LIN {X 0,Y 343.887,Z 716.045,A -85,B 0,C 180,E1 -14281.046,E2 -14281.046} C_VEL
LIN {X 0,Y 344.919,Z 706.382,A -85,B 0,C 180,E1 -14282.219,E2 -14282.219} C_VEL
LIN {X 0,Y 345.964,Z 694.644,A -85,B 0,C 180,E1 -14283.359,E2 -14283.359} C_VEL
LIN {X 0,Y 346.283,Z 691.22,A -85,B 0,C 180,E1 -14283.642,E2 -14283.642} C_VEL
LIN {X 0,Y 344.349,Z 679.11,A -85,B 0,C 180,E1 -14284.621,E2 -14284.621} C_VEL
LIN {X 0,Y 341.376,Z 665.612,A -85,B 0,C 180,E1 -14285.494,E2 -14285.494} C_VEL
LIN {X 0,Y 339.656,Z 658.402,A -85,B 0,C 180,E1 -14285.879,E2 -14285.879} C_VEL
LIN {X 0,Y 339.842,Z 654.272,A -85,B 0,C 180,E1 -14289.417,E2 -14289.417} C_VEL
LIN {X 0,Y 340.111,Z 649.95,A -85,B 0,C 180,E1 -14293.184,E2 -14293.184} C_VEL
LIN {X 0,Y 340.493,Z 645.812,A -85,B 0,C 180,E1 -14296.876,E2 -14296.876} C_VEL
LIN {X 0,Y 340.727,Z 642.044,A -85,B 0,C 180,E1 -14300.502,E2 -14300.502} C_VEL
LIN {X 0,Y 341.051,Z 642.005,A -85,B 0,C 180,E1 -14302.897,E2 -14302.897} C_VEL
LIN {X 0,Y 341.173,Z 641.984,A -85,B 0,C 180,E1 -14307.638,E2 -14307.638} C_VEL
LIN {X 0,Y 341.3,Z 641.968,A -85,B 0,C 180,E1 -14310,E2 -14310} C_VEL
LIN {X 0,Y 341.172,Z 641.985,A -85,B 0,C 180,E1 -14312.361,E2 -14312.361} C_VEL
LIN {X 0,Y 341.028,Z 642.002,A -85,B 0,C 180,E1 -14315.914,E2 -14315.914} C_VEL
LIN {X 0,Y 340.866,Z 642.023,A -85,B 0,C 180,E1 -14318.298,E2 -14318.298} C_VEL
LIN {X 0,Y 340.336,Z 642.088,A -85,B 0,C 180,E1 -14321.917,E2 -14321.917} C_VEL
LIN {X 0,Y 340.189,Z 642.443,A -85,B 0,C 180,E1 -14322.528,E2 -14322.528} C_VEL
LIN {X 0,Y 339.825,Z 648.464,A -85,B 0,C 180,E1 -14326.83,E2 -14326.83} C_VEL
LIN {X 0,Y 339.592,Z 653.752,A -85,B 0,C 180,E1 -14330.598,E2 -14330.598} C_VEL
LIN {X 0,Y 339.509,Z 657.449,A -85,B 0,C 180,E1 -14333.241,E2 -14333.241} C_VEL
LIN {X 0,Y 342.868,Z 671.995,A -85,B 0,C 180,E1 -14334.04,E2 -14334.04} C_VEL
LIN {X 0,Y 345.151,Z 683.532,A -85,B 0,C 180,E1 -14334.867,E2 -14334.867} C_VEL
LIN {X 0,Y 346.164,Z 690.83,A -85,B 0,C 180,E1 -14335.477,E2 -14335.477} C_VEL
LIN {X 0,Y 345.207,Z 701.967,A -85,B 0,C 180,E1 -14336.467,E2 -14336.467} C_VEL
LIN {X 0,Y 344.102,Z 712.788,A -85,B 0,C 180,E1 -14337.687,E2 -14337.687} C_VEL
LIN {X 0,Y 342.966,Z 723.402,A -85,B 0,C 180,E1 -14339.183,E2 -14339.183} C_VEL
LIN {X 0,Y 341.993,Z 731.641,A -85,B 0,C 180,E1 -14340.609,E2 -14340.609} C_VEL
LIN {X 0,Y 341.029,Z 740,A -85,B 0,C 180,E1 -14342.398,E2 -14342.398} C_VEL
LIN {X 0,Y 340.265,Z 747.036,A -85,B 0,C 180,E1 -14344.291,E2 -14344.291} C_VEL
LIN {X 0,Y 339.695,Z 752.623,A -85,B 0,C 180,E1 -14346.208,E2 -14346.208} C_VEL
LIN {X 0,Y 339.249,Z 757.368,A -85,B 0,C 180,E1 -14348.424,E2 -14348.424} C_VEL
LIN {X 0,Y 338.966,Z 759.987,A -85,B 0,C 180,E1 -14350.18,E2 -14350.18} C_VEL
LIN {X 0,Y 338.177,Z 761.122,A -85,B 0,C 180,E1 -14351.156,E2 -14351.156} C_VEL
LIN {X 0,Y 335.209,Z 762.337,A -85,B 0,C 180,E1 -14352.752,E2 -14352.752} C_VEL
LIN {X 0,Y 332.789,Z 762.794,A -85,B 0,C 180,E1 -14354.052,E2 -14354.052} C_VEL
LIN {X 0,Y 331.794,Z 762.817,A -85,B 0,C 180,E1 -14355.061,E2 -14355.061} C_VEL
LIN {X 0,Y 331.734,Z 762.729,A -85,B 0,C 180,E1 -14355.402,E2 -14355.402} C_VEL
LIN {X 0,Y 331.941,Z 761.386,A -85,B 0,C 180,E1 -14357.819,E2 -14357.819} C_VEL
LIN {X 0,Y 332.191,Z 759.33,A -85,B 0,C 180,E1 -14359.607,E2 -14359.607} C_VEL
LIN {X 0,Y 332.629,Z 756.285,A -85,B 0,C 180,E1 -14361.421,E2 -14361.421} C_VEL
LIN {X 0,Y 333.184,Z 752.093,A -85,B 0,C 180,E1 -14363.277,E2 -14363.277} C_VEL
LIN {X 0,Y 334.084,Z 745.842,A -85,B 0,C 180,E1 -14365.39,E2 -14365.39} C_VEL
LIN {X 0,Y 335.2,Z 738.06,A -85,B 0,C 180,E1 -14367.407,E2 -14367.407} C_VEL
LIN {X 0,Y 336.361,Z 730.689,A -85,B 0,C 180,E1 -14368.942,E2 -14368.942} C_VEL
LIN {X 0,Y 337.701,Z 721.438,A -85,B 0,C 180,E1 -14370.522,E2 -14370.522} C_VEL
LIN {X 0,Y 339.034,Z 711.873,A -85,B 0,C 180,E1 -14371.838,E2 -14371.838} C_VEL
LIN {X 0,Y 340.374,Z 700.364,A -85,B 0,C 180,E1 -14373.111,E2 -14373.111} C_VEL
LIN {X 0,Y 341.026,Z 692.815,A -85,B 0,C 180,E1 -14373.804,E2 -14373.804} C_VEL
LIN {X 0,Y 339.014,Z 680.497,A -85,B 0,C 180,E1 -14374.932,E2 -14374.932} C_VEL
LIN {X 0,Y 335.765,Z 667.742,A -85,B 0,C 180,E1 -14375.943,E2 -14375.943} C_VEL
LIN {X 0,Y 332.789,Z 658.389,A -85,B 0,C 180,E1 -14376.591,E2 -14376.591} C_VEL
LIN {X 0,Y 332.987,Z 653.339,A -85,B 0,C 180,E1 -14380.263,E2 -14380.263} C_VEL
LIN {X 0,Y 333.147,Z 649.771,A -85,B 0,C 180,E1 -14382.822,E2 -14382.822} C_VEL
LIN {X 0,Y 333.525,Z 644.51,A -85,B 0,C 180,E1 -14386.597,E2 -14386.597} C_VEL
LIN {X 0,Y 333.508,Z 642.948,A -85,B 0,C 180,E1 -14387.835,E2 -14387.835} C_VEL
LIN {X 0,Y 333.925,Z 642.894,A -85,B 0,C 180,E1 -14391.563,E2 -14391.563} C_VEL
LIN {X 0,Y 334.012,Z 642.883,A -85,B 0,C 180,E1 -14393.961,E2 -14393.961} C_VEL
LIN {X 0,Y 334.104,Z 642.869,A -85,B 0,C 180,E1 -14397.589,E2 -14397.589} C_VEL
LIN {X 0,Y 334.264,Z 642.85,A -85,B 0,C 180,E1 -14400,E2 -14400} C_VEL
LIN {X 0,Y 334.104,Z 642.87,A -85,B 0,C 180,E1 -14402.411,E2 -14402.411} C_VEL
LIN {X 0,Y 334.022,Z 642.879,A -85,B 0,C 180,E1 -14407.253,E2 -14407.253} C_VEL
LIN {X 0,Y 333.83,Z 642.903,A -85,B 0,C 180,E1 -14410.922,E2 -14410.922} C_VEL
LIN {X 0,Y 333.804,Z 642.904,A -85,B 0,C 180,E1 -14414.634,E2 -14414.634} C_VEL
LIN {X 0,Y 333.793,Z 642.906,A -85,B 0,C 180,E1 -14418.656,E2 -14418.656} C_VEL
LIN {X 0,Y 333.689,Z 642.921,A -85,B 0,C 180,E1 -14422.278,E2 -14422.278} C_VEL
LIN {X 0,Y 333.733,Z 642.913,A -85,B 0,C 180,E1 -14426.247,E2 -14426.247} C_VEL
LIN {X 0,Y 333.708,Z 642.916,A -85,B 0,C 180,E1 -14428.972,E2 -14428.972} C_VEL
LIN {X 0,Y 333.64,Z 642.926,A -85,B 0,C 180,E1 -14432.587,E2 -14432.587} C_VEL
LIN {X 0,Y 333.674,Z 642.922,A -85,B 0,C 180,E1 -14436.139,E2 -14436.139} C_VEL
LIN {X 0,Y 333.644,Z 642.927,A -85,B 0,C 180,E1 -14439.193,E2 -14439.193} C_VEL
LIN {X 0,Y 333.63,Z 642.927,A -85,B 0,C 180,E1 -14442.501,E2 -14442.501} C_VEL
LIN {X 0,Y 333.699,Z 643.1,A -85,B 0,C 180,E1 -14446.659,E2 -14446.659} C_VEL
LIN {X 0,Y 334.54,Z 647.77,A -85,B 0,C 180,E1 -14450.154,E2 -14450.154} C_VEL
LIN {X 0,Y 335.04,Z 651.547,A -85,B 0,C 180,E1 -14452.855,E2 -14452.855} C_VEL
LIN {X 0,Y 335.093,Z 654.529,A -85,B 0,C 180,E1 -14454.881,E2 -14454.881} C_VEL
LIN {X 0,Y 334.469,Z 659.801,A -85,B 0,C 180,E1 -14458.312,E2 -14458.312} C_VEL
LIN {X 0,Y 334.02,Z 664.14,A -85,B 0,C 180,E1 -14461.058,E2 -14461.058} C_VEL
LIN {X 0,Y 333.409,Z 670.604,A -85,B 0,C 180,E1 -14465.066,E2 -14465.066} C_VEL
LIN {X 0,Y 333.052,Z 675.105,A -85,B 0,C 180,E1 -14467.763,E2 -14467.763} C_VEL
LIN {X 0,Y 336.355,Z 689.153,A -85,B 0,C 180,E1 -14468.626,E2 -14468.626} C_VEL
LIN {X 0,Y 338.206,Z 701.155,A -85,B 0,C 180,E1 -14469.526,E2 -14469.526} C_VEL
LIN {X 0,Y 339.301,Z 713.613,A -85,B 0,C 180,E1 -14470.646,E2 -14470.646} C_VEL
LIN {X 0,Y 339.303,Z 718.335,A -85,B 0,C 180,E1 -14471.117,E2 -14471.117} C_VEL
LIN {X 0,Y 337.949,Z 729.167,A -85,B 0,C 180,E1 -14472.294,E2 -14472.294} C_VEL
LIN {X 0,Y 336.552,Z 740.044,A -85,B 0,C 180,E1 -14473.798,E2 -14473.798} C_VEL
LIN {X 0,Y 335.251,Z 749.542,A -85,B 0,C 180,E1 -14475.431,E2 -14475.431} C_VEL
LIN {X 0,Y 334.107,Z 757.933,A -85,B 0,C 180,E1 -14477.241,E2 -14477.241} C_VEL
LIN {X 0,Y 333.243,Z 764.702,A -85,B 0,C 180,E1 -14479.059,E2 -14479.059} C_VEL
LIN {X 0,Y 332.621,Z 770.129,A -85,B 0,C 180,E1 -14480.883,E2 -14480.883} C_VEL
LIN {X 0,Y 332.157,Z 775.843,A -85,B 0,C 180,E1 -14483.318,E2 -14483.318} C_VEL
LIN {X 0,Y 332.012,Z 779.038,A -85,B 0,C 180,E1 -14485.143,E2 -14485.143} C_VEL
LIN {X 0,Y 332,Z 780.628,A -85,B 0,C 180,E1 -14486.359,E2 -14486.359} C_VEL
LIN {X 0,Y 331.916,Z 781.79,A -85,B 0,C 180,E1 -14487.573,E2 -14487.573} C_VEL
LIN {X 0,Y 331.925,Z 782.506,A -85,B 0,C 180,E1 -14488.787,E2 -14488.787} C_VEL
LIN {X 0,Y 331.972,Z 782.827,A -85,B 0,C 180,E1 -14490.001,E2 -14490.001} C_VEL
LIN {X 0,Y 331.922,Z 782.752,A -85,B 0,C 180,E1 -14491.214,E2 -14491.214} C_VEL
LIN {X 0,Y 331.914,Z 782.275,A -85,B 0,C 180,E1 -14492.428,E2 -14492.428} C_VEL
LIN {X 0,Y 331.998,Z 781.36,A -85,B 0,C 180,E1 -14493.642,E2 -14493.642} C_VEL
LIN {X 0,Y 332.1,Z 778.315,A -85,B 0,C 180,E1 -14496.074,E2 -14496.074} C_VEL
LIN {X 0,Y 332.377,Z 774.864,A -85,B 0,C 180,E1 -14497.9,E2 -14497.9} C_VEL
LIN {X 0,Y 332.83,Z 770.338,A -85,B 0,C 180,E1 -14499.726,E2 -14499.726} C_VEL
LIN {X 0,Y 333.53,Z 764.63,A -85,B 0,C 180,E1 -14501.548,E2 -14501.548} C_VEL
LIN {X 0,Y 334.595,Z 757.51,A -85,B 0,C 180,E1 -14503.359,E2 -14503.359} C_VEL
LIN {X 0,Y 335.905,Z 748.669,A -85,B 0,C 180,E1 -14505.161,E2 -14505.161} C_VEL
LIN {X 0,Y 337.134,Z 738.987,A -85,B 0,C 180,E1 -14506.766,E2 -14506.766} C_VEL
LIN {X 0,Y 338.547,Z 728.563,A -85,B 0,C 180,E1 -14508.143,E2 -14508.143} C_VEL
LIN {X 0,Y 339.976,Z 717.451,A -85,B 0,C 180,E1 -14509.315,E2 -14509.315} C_VEL
LIN {X 0,Y 339.221,Z 705.114,A -85,B 0,C 180,E1 -14510.483,E2 -14510.483} C_VEL
LIN {X 0,Y 337.175,Z 692.156,A -85,B 0,C 180,E1 -14511.525,E2 -14511.525} C_VEL
LIN {X 0,Y 334.348,Z 680.067,A -85,B 0,C 180,E1 -14512.349,E2 -14512.349} C_VEL
LIN {X 0,Y 333.232,Z 675.513,A -85,B 0,C 180,E1 -14512.642,E2 -14512.642} C_VEL
LIN {X 0,Y 333.811,Z 668.75,A -85,B 0,C 180,E1 -14516.915,E2 -14516.915} C_VEL
LIN {X 0,Y 334.465,Z 663.296,A -85,B 0,C 180,E1 -14520.512,E2 -14520.512} C_VEL
LIN {X 0,Y 334.971,Z 659.603,A -85,B 0,C 180,E1 -14523.059,E2 -14523.059} C_VEL
LIN {X 0,Y 335.311,Z 655.648,A -85,B 0,C 180,E1 -14525.936,E2 -14525.936} C_VEL
LIN {X 0,Y 335.104,Z 651.672,A -85,B 0,C 180,E1 -14529.105,E2 -14529.105} C_VEL
LIN {X 0,Y 334.499,Z 647.664,A -85,B 0,C 180,E1 -14532.662,E2 -14532.662} C_VEL
LIN {X 0,Y 333.883,Z 644.312,A -85,B 0,C 180,E1 -14536.002,E2 -14536.002} C_VEL
LIN {X 0,Y 333.643,Z 642.928,A -85,B 0,C 180,E1 -14537.619,E2 -14537.619} C_VEL
LIN {X 0,Y 333.654,Z 642.927,A -85,B 0,C 180,E1 -14541.202,E2 -14541.202} C_VEL
LIN {X 0,Y 333.678,Z 642.924,A -85,B 0,C 180,E1 -14543.861,E2 -14543.861} C_VEL
LIN {X 0,Y 333.645,Z 642.925,A -85,B 0,C 180,E1 -14547.413,E2 -14547.413} C_VEL
LIN {X 0,Y 333.692,Z 642.92,A -85,B 0,C 180,E1 -14551.026,E2 -14551.026} C_VEL
LIN {X 0,Y 333.737,Z 642.911,A -85,B 0,C 180,E1 -14553.754,E2 -14553.754} C_VEL
LIN {X 0,Y 333.721,Z 642.917,A -85,B 0,C 180,E1 -14557.914,E2 -14557.914} C_VEL
LIN {X 0,Y 333.796,Z 642.908,A -85,B 0,C 180,E1 -14561.59,E2 -14561.59} C_VEL
LIN {X 0,Y 333.81,Z 642.907,A -85,B 0,C 180,E1 -14565.577,E2 -14565.577} C_VEL
LIN {X 0,Y 333.836,Z 642.903,A -85,B 0,C 180,E1 -14569.078,E2 -14569.078} C_VEL
LIN {X 0,Y 334.027,Z 642.878,A -85,B 0,C 180,E1 -14572.748,E2 -14572.748} C_VEL
LIN {X 0,Y 333.813,Z 642.906,A -85,B 0,C 180,E1 -14575.169,E2 -14575.169} C_VEL
LIN {X 0,Y 334.107,Z 642.867,A -85,B 0,C 180,E1 -14577.589,E2 -14577.589} C_VEL
LIN {X 0,Y 334.249,Z 642.851,A -85,B 0,C 180,E1 -14580,E2 -14580} C_VEL
LIN {X 0,Y 334.109,Z 642.871,A -85,B 0,C 180,E1 -14582.411,E2 -14582.411} C_VEL
LIN {X 0,Y 333.851,Z 642.903,A -85,B 0,C 180,E1 -14583.621,E2 -14583.621} C_VEL
LIN {X 0,Y 333.874,Z 643.33,A -85,B 0,C 180,E1 -14584.83,E2 -14584.83} C_VEL
LIN {X 0,Y 334.288,Z 645.219,A -85,B 0,C 180,E1 -14587.247,E2 -14587.247} C_VEL
LIN {X 0,Y 334.222,Z 647.299,A -85,B 0,C 180,E1 -14589.685,E2 -14589.685} C_VEL
LIN {X 0,Y 333.822,Z 650.713,A -85,B 0,C 180,E1 -14593.39,E2 -14593.39} C_VEL
LIN {X 0,Y 333.411,Z 654.396,A -85,B 0,C 180,E1 -14597.164,E2 -14597.164} C_VEL
LIN {X 0,Y 333.052,Z 658.348,A -85,B 0,C 180,E1 -14601.022,E2 -14601.022} C_VEL
LIN {X 0,Y 332.945,Z 659.916,A -85,B 0,C 180,E1 -14602.454,E2 -14602.454} C_VEL
LIN {X 0,Y 334.924,Z 665.893,A -85,B 0,C 180,E1 -14602.866,E2 -14602.866} C_VEL
LIN {X 0,Y 338.155,Z 677.169,A -85,B 0,C 180,E1 -14603.746,E2 -14603.746} C_VEL
LIN {X 0,Y 340.197,Z 686.586,A -85,B 0,C 180,E1 -14604.577,E2 -14604.577} C_VEL
LIN {X 0,Y 341.253,Z 694.62,A -85,B 0,C 180,E1 -14605.356,E2 -14605.356} C_VEL
LIN {X 0,Y 339.972,Z 705.362,A -85,B 0,C 180,E1 -14606.389,E2 -14606.389} C_VEL
LIN {X 0,Y 338.659,Z 715.933,A -85,B 0,C 180,E1 -14607.667,E2 -14607.667} C_VEL
LIN {X 0,Y 337.213,Z 725.82,A -85,B 0,C 180,E1 -14609.159,E2 -14609.159} C_VEL
LIN {X 0,Y 335.819,Z 735.103,A -85,B 0,C 180,E1 -14610.902,E2 -14610.902} C_VEL
LIN {X 0,Y 334.778,Z 742.114,A -85,B 0,C 180,E1 -14612.532,E2 -14612.532} C_VEL
LIN {X 0,Y 333.856,Z 748.201,A -85,B 0,C 180,E1 -14614.272,E2 -14614.272} C_VEL
LIN {X 0,Y 333.081,Z 753.553,A -85,B 0,C 180,E1 -14616.214,E2 -14616.214} C_VEL
LIN {X 0,Y 332.489,Z 758.289,A -85,B 0,C 180,E1 -14618.547,E2 -14618.547} C_VEL
LIN {X 0,Y 332.005,Z 761.528,A -85,B 0,C 180,E1 -14621.012,E2 -14621.012} C_VEL
LIN {X 0,Y 331.866,Z 762.755,A -85,B 0,C 180,E1 -14622.662,E2 -14622.662} C_VEL
LIN {X 0,Y 331.753,Z 763.207,A -85,B 0,C 180,E1 -14624.354,E2 -14624.354} C_VEL
LIN {X 0,Y 331.756,Z 762.88,A -85,B 0,C 180,E1 -14626.077,E2 -14626.077} C_VEL
LIN {X 0,Y 331.862,Z 761.721,A -85,B 0,C 180,E1 -14627.835,E2 -14627.835} C_VEL
LIN {X 0,Y 332.08,Z 759.647,A -85,B 0,C 180,E1 -14629.631,E2 -14629.631} C_VEL
LIN {X 0,Y 332.375,Z 756.523,A -85,B 0,C 180,E1 -14631.477,E2 -14631.477} C_VEL
LIN {X 0,Y 332.922,Z 751.114,A -85,B 0,C 180,E1 -14633.766,E2 -14633.766} C_VEL
LIN {X 0,Y 333.541,Z 745.111,A -85,B 0,C 180,E1 -14635.691,E2 -14635.691} C_VEL
LIN {X 0,Y 334.396,Z 737.874,A -85,B 0,C 180,E1 -14637.519,E2 -14637.519} C_VEL
LIN {X 0,Y 335.431,Z 729.564,A -85,B 0,C 180,E1 -14639.209,E2 -14639.209} C_VEL
LIN {X 0,Y 336.509,Z 720.29,A -85,B 0,C 180,E1 -14640.747,E2 -14640.747} C_VEL
LIN {X 0,Y 337.656,Z 710.407,A -85,B 0,C 180,E1 -14642.075,E2 -14642.075} C_VEL
LIN {X 0,Y 338.721,Z 699.199,A -85,B 0,C 180,E1 -14643.282,E2 -14643.282} C_VEL
LIN {X 0,Y 339.263,Z 690.604,A -85,B 0,C 180,E1 -14644.048,E2 -14644.048} C_VEL
LIN {X 0,Y 337.079,Z 678.122,A -85,B 0,C 180,E1 -14645.071,E2 -14645.071} C_VEL
LIN {X 0,Y 334.142,Z 665.017,A -85,B 0,C 180,E1 -14645.93,E2 -14645.93} C_VEL
LIN {X 0,Y 332.598,Z 658.588,A -85,B 0,C 180,E1 -14646.292,E2 -14646.292} C_VEL
LIN {X 0,Y 332.831,Z 654.037,A -85,B 0,C 180,E1 -14650.253,E2 -14650.253} C_VEL
LIN {X 0,Y 333.131,Z 649.745,A -85,B 0,C 180,E1 -14654.082,E2 -14654.082} C_VEL
LIN {X 0,Y 333.411,Z 646.98,A -85,B 0,C 180,E1 -14656.592,E2 -14656.592} C_VEL
LIN {X 0,Y 333.666,Z 643.014,A -85,B 0,C 180,E1 -14660.299,E2 -14660.299} C_VEL
LIN {X 0,Y 333.994,Z 642.882,A -85,B 0,C 180,E1 -14662.746,E2 -14662.746} C_VEL
LIN {X 0,Y 333.812,Z 642.904,A -85,B 0,C 180,E1 -14665.169,E2 -14665.169} C_VEL
LIN {X 0,Y 334.11,Z 642.864,A -85,B 0,C 180,E1 -14667.588,E2 -14667.588} C_VEL
LIN {X 0,Y 334.251,Z 642.846,A -85,B 0,C 180,E1 -14669.999,E2 -14669.999} C_VEL
LIN {X 0,Y 334.11,Z 642.865,A -85,B 0,C 180,E1 -14672.411,E2 -14672.411} C_VEL
LIN {X 0,Y 333.999,Z 642.878,A -85,B 0,C 180,E1 -14676.039,E2 -14676.039} C_VEL
LIN {X 0,Y 333.787,Z 642.906,A -85,B 0,C 180,E1 -14678.475,E2 -14678.475} C_VEL
LIN {X 0,Y 333.187,Z 642.988,A -85,B 0,C 180,E1 -14682.292,E2 -14682.292} C_VEL
LIN {X 0,Y 332.798,Z 648.01,A -85,B 0,C 180,E1 -14685.934,E2 -14685.934} C_VEL
LIN {X 0,Y 332.662,Z 651.536,A -85,B 0,C 180,E1 -14688.475,E2 -14688.475} C_VEL
LIN {X 0,Y 332.434,Z 656.948,A -85,B 0,C 180,E1 -14692.366,E2 -14692.366} C_VEL
LIN {X 0,Y 332.45,Z 657.693,A -85,B 0,C 180,E1 -14692.857,E2 -14692.857} C_VEL
LIN {X 0,Y 335.759,Z 671.72,A -85,B 0,C 180,E1 -14693.638,E2 -14693.638} C_VEL
LIN {X 0,Y 338.216,Z 684.197,A -85,B 0,C 180,E1 -14694.556,E2 -14694.556} C_VEL
LIN {X 0,Y 339.313,Z 691.71,A -85,B 0,C 180,E1 -14695.207,E2 -14695.207} C_VEL
LIN {X 0,Y 338.268,Z 703.087,A -85,B 0,C 180,E1 -14696.257,E2 -14696.257} C_VEL
LIN {X 0,Y 337.023,Z 714.803,A -85,B 0,C 180,E1 -14697.644,E2 -14697.644} C_VEL
LIN {X 0,Y 335.884,Z 724.714,A -85,B 0,C 180,E1 -14699.109,E2 -14699.109} C_VEL
LIN {X 0,Y 334.75,Z 734.035,A -85,B 0,C 180,E1 -14700.83,E2 -14700.83} C_VEL
LIN {X 0,Y 333.858,Z 741.937,A -85,B 0,C 180,E1 -14702.644,E2 -14702.644} C_VEL
LIN {X 0,Y 333.077,Z 748.729,A -85,B 0,C 180,E1 -14704.623,E2 -14704.623} C_VEL
LIN {X 0,Y 332.501,Z 753.912,A -85,B 0,C 180,E1 -14706.563,E2 -14706.563} C_VEL
LIN {X 0,Y 332.149,Z 757.763,A -85,B 0,C 180,E1 -14708.474,E2 -14708.474} C_VEL
LIN {X 0,Y 331.848,Z 760.418,A -85,B 0,C 180,E1 -14710.322,E2 -14710.322} C_VEL
LIN {X 0,Y 331.678,Z 762.405,A -85,B 0,C 180,E1 -14712.691,E2 -14712.691} C_VEL
LIN {X 0,Y 331.719,Z 762.87,A -85,B 0,C 180,E1 -14714.358,E2 -14714.358} C_VEL
LIN {X 0,Y 331.734,Z 762.729,A -85,B 0,C 180,E1 -14715.402,E2 -14715.402} C_VEL
LIN {X 0,Y 331.141,Z 762.46,A -85,B 0,C 180,E1 -14716.416,E2 -14716.416} C_VEL
LIN {X 0,Y 328.43,Z 761.437,A -85,B 0,C 180,E1 -14718.064,E2 -14718.064} C_VEL
LIN {X 0,Y 326.193,Z 760.057,A -85,B 0,C 180,E1 -14719.384,E2 -14719.384} C_VEL
LIN {X 0,Y 325.35,Z 758.678,A -85,B 0,C 180,E1 -14720.389,E2 -14720.389} C_VEL
LIN {X 0,Y 325.346,Z 758.123,A -85,B 0,C 180,E1 -14720.725,E2 -14720.725} C_VEL
LIN {X 0,Y 325.989,Z 753.834,A -85,B 0,C 180,E1 -14722.908,E2 -14722.908} C_VEL
LIN {X 0,Y 326.729,Z 748.798,A -85,B 0,C 180,E1 -14724.823,E2 -14724.823} C_VEL
LIN {X 0,Y 327.748,Z 742.304,A -85,B 0,C 180,E1 -14726.749,E2 -14726.749} C_VEL
LIN {X 0,Y 329.093,Z 734.103,A -85,B 0,C 180,E1 -14728.673,E2 -14728.673} C_VEL
LIN {X 0,Y 330.429,Z 725.241,A -85,B 0,C 180,E1 -14730.347,E2 -14730.347} C_VEL
LIN {X 0,Y 331.967,Z 714.941,A -85,B 0,C 180,E1 -14731.897,E2 -14731.897} C_VEL
LIN {X 0,Y 333.399,Z 704.029,A -85,B 0,C 180,E1 -14733.219,E2 -14733.219} C_VEL
LIN {X 0,Y 334.446,Z 694.487,A -85,B 0,C 180,E1 -14734.149,E2 -14734.149} C_VEL
LIN {X 0,Y 332.802,Z 683.728,A -85,B 0,C 180,E1 -14735.2,E2 -14735.2} C_VEL
LIN {X 0,Y 329.742,Z 670.964,A -85,B 0,C 180,E1 -14736.278,E2 -14736.278} C_VEL
LIN {X 0,Y 325.783,Z 658.559,A -85,B 0,C 180,E1 -14737.222,E2 -14737.222} C_VEL
LIN {X 0,Y 326.081,Z 652.738,A -85,B 0,C 180,E1 -14741.498,E2 -14741.498} C_VEL
LIN {X 0,Y 326.42,Z 647.051,A -85,B 0,C 180,E1 -14745.664,E2 -14745.664} C_VEL
LIN {X 0,Y 326.503,Z 643.819,A -85,B 0,C 180,E1 -14748.122,E2 -14748.122} C_VEL
LIN {X 0,Y 326.867,Z 643.773,A -85,B 0,C 180,E1 -14751.508,E2 -14751.508} C_VEL
LIN {X 0,Y 326.986,Z 643.758,A -85,B 0,C 180,E1 -14753.831,E2 -14753.831} C_VEL
LIN {X 0,Y 327.045,Z 643.748,A -85,B 0,C 180,E1 -14757.537,E2 -14757.537} C_VEL
LIN {X 0,Y 327.215,Z 643.728,A -85,B 0,C 180,E1 -14760,E2 -14760} C_VEL
LIN {X 0,Y 327.045,Z 643.749,A -85,B 0,C 180,E1 -14762.463,E2 -14762.463} C_VEL
LIN {X 0,Y 326.993,Z 643.754,A -85,B 0,C 180,E1 -14766.169,E2 -14766.169} C_VEL
LIN {X 0,Y 326.911,Z 643.766,A -85,B 0,C 180,E1 -14768.655,E2 -14768.655} C_VEL
LIN {X 0,Y 326.731,Z 643.786,A -85,B 0,C 180,E1 -14772.421,E2 -14772.421} C_VEL
LIN {X 0,Y 326.75,Z 643.785,A -85,B 0,C 180,E1 -14774.958,E2 -14774.958} C_VEL
LIN {X 0,Y 326.73,Z 643.785,A -85,B 0,C 180,E1 -14778.839,E2 -14778.839} C_VEL
LIN {X 0,Y 326.617,Z 643.802,A -85,B 0,C 180,E1 -14782.788,E2 -14782.788} C_VEL
LIN {X 0,Y 326.687,Z 643.792,A -85,B 0,C 180,E1 -14785.484,E2 -14785.484} C_VEL
LIN {X 0,Y 326.658,Z 643.797,A -85,B 0,C 180,E1 -14789.659,E2 -14789.659} C_VEL
LIN {X 0,Y 326.604,Z 643.803,A -85,B 0,C 180,E1 -14794.02,E2 -14794.02} C_VEL
LIN {X 0,Y 326.625,Z 643.799,A -85,B 0,C 180,E1 -14797.239,E2 -14797.239} C_VEL
LIN {X 0,Y 326.575,Z 643.807,A -85,B 0,C 180,E1 -14801.132,E2 -14801.132} C_VEL
LIN {X 0,Y 326.527,Z 643.813,A -85,B 0,C 180,E1 -14804.744,E2 -14804.744} C_VEL
LIN {X 0,Y 326.622,Z 643.943,A -85,B 0,C 180,E1 -14806.38,E2 -14806.38} C_VEL
LIN {X 0,Y 327.465,Z 648.546,A -85,B 0,C 180,E1 -14809.921,E2 -14809.921} C_VEL
LIN {X 0,Y 327.969,Z 652.011,A -85,B 0,C 180,E1 -14812.455,E2 -14812.455} C_VEL
LIN {X 0,Y 328.084,Z 655.177,A -85,B 0,C 180,E1 -14814.664,E2 -14814.664} C_VEL
LIN {X 0,Y 327.428,Z 660.592,A -85,B 0,C 180,E1 -14818.274,E2 -14818.274} C_VEL
LIN {X 0,Y 326.83,Z 666.118,A -85,B 0,C 180,E1 -14821.842,E2 -14821.842} C_VEL
LIN {X 0,Y 326.207,Z 672.453,A -85,B 0,C 180,E1 -14825.837,E2 -14825.837} C_VEL
LIN {X 0,Y 326.072,Z 674.537,A -85,B 0,C 180,E1 -14827.131,E2 -14827.131} C_VEL
LIN {X 0,Y 329.583,Z 689.409,A -85,B 0,C 180,E1 -14828.103,E2 -14828.103} C_VEL
LIN {X 0,Y 331.348,Z 700.31,A -85,B 0,C 180,E1 -14828.949,E2 -14828.949} C_VEL
LIN {X 0,Y 332.452,Z 712.423,A -85,B 0,C 180,E1 -14830.058,E2 -14830.058} C_VEL
LIN {X 0,Y 332.612,Z 718.831,A -85,B 0,C 180,E1 -14830.723,E2 -14830.723} C_VEL
LIN {X 0,Y 331.209,Z 729.47,A -85,B 0,C 180,E1 -14831.921,E2 -14831.921} C_VEL
LIN {X 0,Y 329.707,Z 740.469,A -85,B 0,C 180,E1 -14833.492,E2 -14833.492} C_VEL
LIN {X 0,Y 328.366,Z 749.656,A -85,B 0,C 180,E1 -14835.118,E2 -14835.118} C_VEL
LIN {X 0,Y 327.178,Z 757.977,A -85,B 0,C 180,E1 -14836.966,E2 -14836.966} C_VEL
LIN {X 0,Y 326.242,Z 764.703,A -85,B 0,C 180,E1 -14838.821,E2 -14838.821} C_VEL
LIN {X 0,Y 325.588,Z 770.08,A -85,B 0,C 180,E1 -14840.684,E2 -14840.684} C_VEL
LIN {X 0,Y 325.074,Z 775.517,A -85,B 0,C 180,E1 -14843.171,E2 -14843.171} C_VEL
LIN {X 0,Y 324.922,Z 778.742,A -85,B 0,C 180,E1 -14845.037,E2 -14845.037} C_VEL
LIN {X 0,Y 324.906,Z 780.348,A -85,B 0,C 180,E1 -14846.28,E2 -14846.28} C_VEL
LIN {X 0,Y 324.836,Z 781.535,A -85,B 0,C 180,E1 -14847.521,E2 -14847.521} C_VEL
LIN {X 0,Y 324.833,Z 782.272,A -85,B 0,C 180,E1 -14848.761,E2 -14848.761} C_VEL
LIN {X 0,Y 324.877,Z 782.607,A -85,B 0,C 180,E1 -14850.001,E2 -14850.001} C_VEL
LIN {X 0,Y 324.831,Z 782.546,A -85,B 0,C 180,E1 -14851.24,E2 -14851.24} C_VEL
LIN {X 0,Y 324.835,Z 782.09,A -85,B 0,C 180,E1 -14852.481,E2 -14852.481} C_VEL
LIN {X 0,Y 324.903,Z 781.193,A -85,B 0,C 180,E1 -14853.721,E2 -14853.721} C_VEL
LIN {X 0,Y 325.041,Z 778.184,A -85,B 0,C 180,E1 -14856.207,E2 -14856.207} C_VEL
LIN {X 0,Y 325.326,Z 774.771,A -85,B 0,C 180,E1 -14858.073,E2 -14858.073} C_VEL
LIN {X 0,Y 325.813,Z 770.288,A -85,B 0,C 180,E1 -14859.937,E2 -14859.937} C_VEL
LIN {X 0,Y 326.551,Z 764.618,A -85,B 0,C 180,E1 -14861.798,E2 -14861.798} C_VEL
LIN {X 0,Y 327.671,Z 757.565,A -85,B 0,C 180,E1 -14863.647,E2 -14863.647} C_VEL
LIN {X 0,Y 329.033,Z 748.778,A -85,B 0,C 180,E1 -14865.486,E2 -14865.486} C_VEL
LIN {X 0,Y 330.233,Z 739.838,A -85,B 0,C 180,E1 -14867.015,E2 -14867.015} C_VEL
LIN {X 0,Y 331.835,Z 728.887,A -85,B 0,C 180,E1 -14868.524,E2 -14868.524} C_VEL
LIN {X 0,Y 333.278,Z 717.942,A -85,B 0,C 180,E1 -14869.719,E2 -14869.719} C_VEL
LIN {X 0,Y 332.559,Z 705.976,A -85,B 0,C 180,E1 -14870.904,E2 -14870.904} C_VEL
LIN {X 0,Y 330.707,Z 693.709,A -85,B 0,C 180,E1 -14871.948,E2 -14871.948} C_VEL
LIN {X 0,Y 327.622,Z 680.638,A -85,B 0,C 180,E1 -14872.895,E2 -14872.895} C_VEL
LIN {X 0,Y 326.214,Z 675.258,A -85,B 0,C 180,E1 -14873.27,E2 -14873.27} C_VEL
LIN {X 0,Y 326.886,Z 668.713,A -85,B 0,C 180,E1 -14877.533,E2 -14877.533} C_VEL
LIN {X 0,Y 327.648,Z 662.626,A -85,B 0,C 180,E1 -14881.704,E2 -14881.704} C_VEL
LIN {X 0,Y 328.057,Z 659.644,A -85,B 0,C 180,E1 -14883.849,E2 -14883.849} C_VEL
LIN {X 0,Y 328.3,Z 657.348,A -85,B 0,C 180,E1 -14885.563,E2 -14885.563} C_VEL
LIN {X 0,Y 328.17,Z 653.823,A -85,B 0,C 180,E1 -14888.394,E2 -14888.394} C_VEL
LIN {X 0,Y 327.692,Z 650.119,A -85,B 0,C 180,E1 -14891.672,E2 -14891.672} C_VEL
LIN {X 0,Y 327.089,Z 646.593,A -85,B 0,C 180,E1 -14895.158,E2 -14895.158} C_VEL
LIN {X 0,Y 326.607,Z 643.879,A -85,B 0,C 180,E1 -14898.159,E2 -14898.159} C_VEL
LIN {X 0,Y 326.599,Z 643.805,A -85,B 0,C 180,E1 -14901.388,E2 -14901.388} C_VEL
LIN {X 0,Y 326.621,Z 643.801,A -85,B 0,C 180,E1 -14904.851,E2 -14904.851} C_VEL
LIN {X 0,Y 326.609,Z 643.801,A -85,B 0,C 180,E1 -14907.456,E2 -14907.456} C_VEL
LIN {X 0,Y 326.649,Z 643.797,A -85,B 0,C 180,E1 -14910.34,E2 -14910.34} C_VEL
LIN {X 0,Y 326.692,Z 643.792,A -85,B 0,C 180,E1 -14914.516,E2 -14914.516} C_VEL
LIN {X 0,Y 326.649,Z 643.798,A -85,B 0,C 180,E1 -14918.545,E2 -14918.545} C_VEL
LIN {X 0,Y 326.746,Z 643.785,A -85,B 0,C 180,E1 -14921.178,E2 -14921.178} C_VEL
LIN {X 0,Y 326.765,Z 643.784,A -85,B 0,C 180,E1 -14925.433,E2 -14925.433} C_VEL
LIN {X 0,Y 326.772,Z 643.783,A -85,B 0,C 180,E1 -14928.839,E2 -14928.839} C_VEL
LIN {X 0,Y 326.981,Z 643.754,A -85,B 0,C 180,E1 -14932.59,E2 -14932.59} C_VEL
LIN {X 0,Y 326.78,Z 643.782,A -85,B 0,C 180,E1 -14935.065,E2 -14935.065} C_VEL
LIN {X 0,Y 327.048,Z 643.747,A -85,B 0,C 180,E1 -14937.537,E2 -14937.537} C_VEL
LIN {X 0,Y 327.201,Z 643.729,A -85,B 0,C 180,E1 -14940,E2 -14940} C_VEL
LIN {X 0,Y 327.05,Z 643.75,A -85,B 0,C 180,E1 -14942.463,E2 -14942.463} C_VEL
LIN {X 0,Y 326.802,Z 643.794,A -85,B 0,C 180,E1 -14943.699,E2 -14943.699} C_VEL
LIN {X 0,Y 327.301,Z 646.571,A -85,B 0,C 180,E1 -14947.402,E2 -14947.402} C_VEL
LIN {X 0,Y 327.179,Z 648.667,A -85,B 0,C 180,E1 -14949.895,E2 -14949.895} C_VEL
LIN {X 0,Y 326.781,Z 652.085,A -85,B 0,C 180,E1 -14953.685,E2 -14953.685} C_VEL
LIN {X 0,Y 326.322,Z 655.796,A -85,B 0,C 180,E1 -14957.549,E2 -14957.549} C_VEL
LIN {X 0,Y 325.934,Z 660.076,A -85,B 0,C 180,E1 -14961.809,E2 -14961.809} C_VEL
LIN {X 0,Y 330.66,Z 674.959,A -85,B 0,C 180,E1 -14962.989,E2 -14962.989} C_VEL
LIN {X 0,Y 333.33,Z 686.381,A -85,B 0,C 180,E1 -14964.015,E2 -14964.015} C_VEL
LIN {X 0,Y 334.557,Z 694.648,A -85,B 0,C 180,E1 -14964.843,E2 -14964.843} C_VEL
LIN {X 0,Y 333.742,Z 702.915,A -85,B 0,C 180,E1 -14965.642,E2 -14965.642} C_VEL
LIN {X 0,Y 332.272,Z 714.038,A -85,B 0,C 180,E1 -14966.955,E2 -14966.955} C_VEL
LIN {X 0,Y 330.815,Z 723.792,A -85,B 0,C 180,E1 -14968.382,E2 -14968.382} C_VEL
LIN {X 0,Y 329.359,Z 733.209,A -85,B 0,C 180,E1 -14970.096,E2 -14970.096} C_VEL
LIN {X 0,Y 328.008,Z 741.836,A -85,B 0,C 180,E1 -14972.075,E2 -14972.075} C_VEL
LIN {X 0,Y 326.92,Z 748.446,A -85,B 0,C 180,E1 -14973.983,E2 -14973.983} C_VEL
LIN {X 0,Y 326.24,Z 752.816,A -85,B 0,C 180,E1 -14975.567,E2 -14975.567} C_VEL
LIN {X 0,Y 325.536,Z 757.889,A -85,B 0,C 180,E1 -14977.973,E2 -14977.973} C_VEL
LIN {X 0,Y 325.31,Z 759.446,A -85,B 0,C 180,E1 -14978.945,E2 -14978.945} C_VEL
LIN {X 0,Y 324.939,Z 761.69,A -85,B 0,C 180,E1 -14980.799,E2 -14980.799} C_VEL
LIN {X 0,Y 324.773,Z 763.008,A -85,B 0,C 180,E1 -14982.629,E2 -14982.629} C_VEL
LIN {X 0,Y 324.654,Z 763.435,A -85,B 0,C 180,E1 -14984.408,E2 -14984.408} C_VEL
LIN {X 0,Y 324.659,Z 763.047,A -85,B 0,C 180,E1 -14986.154,E2 -14986.154} C_VEL
LIN {X 0,Y 324.767,Z 761.907,A -85,B 0,C 180,E1 -14987.867,E2 -14987.867} C_VEL
LIN {X 0,Y 324.988,Z 760.037,A -85,B 0,C 180,E1 -14989.551,E2 -14989.551} C_VEL
LIN {X 0,Y 325.24,Z 757.413,A -85,B 0,C 180,E1 -14991.196,E2 -14991.196} C_VEL
LIN {X 0,Y 325.585,Z 753.6,A -85,B 0,C 180,E1 -14993.004,E2 -14993.004} C_VEL
LIN {X 0,Y 326.169,Z 748.251,A -85,B 0,C 180,E1 -14994.964,E2 -14994.964} C_VEL
LIN {X 0,Y 327.013,Z 741.293,A -85,B 0,C 180,E1 -14996.948,E2 -14996.948} C_VEL
LIN {X 0,Y 327.969,Z 733.748,A -85,B 0,C 180,E1 -14998.671,E2 -14998.671} C_VEL
LIN {X 0,Y 329.128,Z 724.371,A -85,B 0,C 180,E1 -15000.409,E2 -15000.409} C_VEL
LIN {X 0,Y 330.377,Z 714.134,A -85,B 0,C 180,E1 -15001.923,E2 -15001.923} C_VEL
LIN {X 0,Y 331.612,Z 702.53,A -85,B 0,C 180,E1 -15003.293,E2 -15003.293} C_VEL
LIN {X 0,Y 332.407,Z 691.725,A -85,B 0,C 180,E1 -15004.314,E2 -15004.314} C_VEL
LIN {X 0,Y 330.387,Z 679.981,A -85,B 0,C 180,E1 -15005.325,E2 -15005.325} C_VEL
LIN {X 0,Y 327.473,Z 666.809,A -85,B 0,C 180,E1 -15006.229,E2 -15006.229} C_VEL
LIN {X 0,Y 325.51,Z 658.835,A -85,B 0,C 180,E1 -15006.668,E2 -15006.668} C_VEL
LIN {X 0,Y 325.724,Z 655.274,A -85,B 0,C 180,E1 -15009.804,E2 -15009.804} C_VEL
LIN {X 0,Y 326.039,Z 650.942,A -85,B 0,C 180,E1 -15013.726,E2 -15013.726} C_VEL
LIN {X 0,Y 326.319,Z 648.15,A -85,B 0,C 180,E1 -15016.295,E2 -15016.295} C_VEL
LIN {X 0,Y 326.615,Z 644.156,A -85,B 0,C 180,E1 -15020.087,E2 -15020.087} C_VEL
LIN {X 0,Y 326.866,Z 643.767,A -85,B 0,C 180,E1 -15021.517,E2 -15021.517} C_VEL
LIN {X 0,Y 326.987,Z 643.751,A -85,B 0,C 180,E1 -15023.83,E2 -15023.83} C_VEL
LIN {X 0,Y 327.05,Z 643.743,A -85,B 0,C 180,E1 -15027.536,E2 -15027.536} C_VEL
LIN {X 0,Y 327.202,Z 643.724,A -85,B 0,C 180,E1 -15029.999,E2 -15029.999} C_VEL
LIN {X 0,Y 327.05,Z 643.744,A -85,B 0,C 180,E1 -15032.463,E2 -15032.463} C_VEL
LIN {X 0,Y 326.949,Z 643.756,A -85,B 0,C 180,E1 -15036.169,E2 -15036.169} C_VEL
LIN {X 0,Y 326.713,Z 643.788,A -85,B 0,C 180,E1 -15038.66,E2 -15038.66} C_VEL
LIN {X 0,Y 326.143,Z 643.858,A -85,B 0,C 180,E1 -15042.286,E2 -15042.286} C_VEL
LIN {X 0,Y 325.72,Z 649.331,A -85,B 0,C 180,E1 -15046.289,E2 -15046.289} C_VEL
LIN {X 0,Y 325.55,Z 652.879,A -85,B 0,C 180,E1 -15048.894,E2 -15048.894} C_VEL
LIN {X 0,Y 325.38,Z 657.775,A -85,B 0,C 180,E1 -15052.45,E2 -15052.45} C_VEL
LIN {X 0,Y 328.633,Z 671.386,A -85,B 0,C 180,E1 -15053.221,E2 -15053.221} C_VEL
LIN {X 0,Y 331.08,Z 683.524,A -85,B 0,C 180,E1 -15054.118,E2 -15054.118} C_VEL
LIN {X 0,Y 332.422,Z 691.686,A -85,B 0,C 180,E1 -15054.846,E2 -15054.846} C_VEL
LIN {X 0,Y 331.423,Z 703.234,A -85,B 0,C 180,E1 -15055.935,E2 -15055.935} C_VEL
LIN {X 0,Y 330.151,Z 714.796,A -85,B 0,C 180,E1 -15057.327,E2 -15057.327} C_VEL
LIN {X 0,Y 328.964,Z 724.88,A -85,B 0,C 180,E1 -15058.845,E2 -15058.845} C_VEL
LIN {X 0,Y 327.825,Z 734.016,A -85,B 0,C 180,E1 -15060.562,E2 -15060.562} C_VEL
LIN {X 0,Y 326.83,Z 742.368,A -85,B 0,C 180,E1 -15062.519,E2 -15062.519} C_VEL
LIN {X 0,Y 326.024,Z 749.036,A -85,B 0,C 180,E1 -15064.516,E2 -15064.516} C_VEL
LIN {X 0,Y 325.489,Z 753.719,A -85,B 0,C 180,E1 -15066.289,E2 -15066.289} C_VEL
LIN {X 0,Y 325.137,Z 757.301,A -85,B 0,C 180,E1 -15068.027,E2 -15068.027} C_VEL
LIN {X 0,Y 324.842,Z 759.853,A -85,B 0,C 180,E1 -15069.659,E2 -15069.659} C_VEL
LIN {X 0,Y 324.716,Z 761.124,A -85,B 0,C 180,E1 -15070.753,E2 -15070.753} C_VEL
LIN {X 0,Y 324.582,Z 762.55,A -85,B 0,C 180,E1 -15072.592,E2 -15072.592} C_VEL
LIN {X 0,Y 324.621,Z 763.067,A -85,B 0,C 180,E1 -15074.402,E2 -15074.402} C_VEL
LIN {X 0,Y 324.689,Z 762.745,A -85,B 0,C 180,E1 -15076.159,E2 -15076.159} C_VEL
LIN {X 0,Y 324.853,Z 761.658,A -85,B 0,C 180,E1 -15077.881,E2 -15077.881} C_VEL
LIN {X 0,Y 325.098,Z 759.844,A -85,B 0,C 180,E1 -15079.568,E2 -15079.568} C_VEL
LIN {X 0,Y 325.346,Z 758.123,A -85,B 0,C 180,E1 -15080.725,E2 -15080.725} C_VEL
LIN {X 0,Y 324.943,Z 756.432,A -85,B 0,C 180,E1 -15081.721,E2 -15081.721} C_VEL
LIN {X 0,Y 322.599,Z 753.328,A -85,B 0,C 180,E1 -15083.339,E2 -15083.339} C_VEL
LIN {X 0,Y 320.382,Z 749.533,A -85,B 0,C 180,E1 -15084.927,E2 -15084.927} C_VEL
LIN {X 0,Y 320.176,Z 746.739,A -85,B 0,C 180,E1 -15085.86,E2 -15085.86} C_VEL
LIN {X 0,Y 321.432,Z 739.064,A -85,B 0,C 180,E1 -15087.98,E2 -15087.98} C_VEL
LIN {X 0,Y 322.702,Z 731.802,A -85,B 0,C 180,E1 -15089.583,E2 -15089.583} C_VEL
LIN {X 0,Y 324.31,Z 721.947,A -85,B 0,C 180,E1 -15091.349,E2 -15091.349} C_VEL
LIN {X 0,Y 325.89,Z 711.013,A -85,B 0,C 180,E1 -15092.9,E2 -15092.9} C_VEL
LIN {X 0,Y 327.337,Z 700.207,A -85,B 0,C 180,E1 -15094.117,E2 -15094.117} C_VEL
LIN {X 0,Y 327.772,Z 695.196,A -85,B 0,C 180,E1 -15094.606,E2 -15094.606} C_VEL
LIN {X 0,Y 325.875,Z 683.266,A -85,B 0,C 180,E1 -15095.81,E2 -15095.81} C_VEL
LIN {X 0,Y 322.707,Z 670.762,A -85,B 0,C 180,E1 -15096.92,E2 -15096.92} C_VEL
LIN {X 0,Y 318.793,Z 658.753,A -85,B 0,C 180,E1 -15097.873,E2 -15097.873} C_VEL
LIN {X 0,Y 319.083,Z 653.183,A -85,B 0,C 180,E1 -15102.04,E2 -15102.04} C_VEL
LIN {X 0,Y 319.472,Z 647.854,A -85,B 0,C 180,E1 -15105.996,E2 -15105.996} C_VEL
LIN {X 0,Y 319.483,Z 644.693,A -85,B 0,C 180,E1 -15108.42,E2 -15108.42} C_VEL
LIN {X 0,Y 319.9,Z 644.642,A -85,B 0,C 180,E1 -15112.425,E2 -15112.425} C_VEL
LIN {X 0,Y 319.745,Z 644.659,A -85,B 0,C 180,E1 -15114.956,E2 -15114.956} C_VEL
LIN {X 0,Y 319.989,Z 644.627,A -85,B 0,C 180,E1 -15117.482,E2 -15117.482} C_VEL
LIN {X 0,Y 320.166,Z 644.606,A -85,B 0,C 180,E1 -15120,E2 -15120} C_VEL
LIN {X 0,Y 319.989,Z 644.628,A -85,B 0,C 180,E1 -15122.518,E2 -15122.518} C_VEL
LIN {X 0,Y 319.948,Z 644.632,A -85,B 0,C 180,E1 -15126.306,E2 -15126.306} C_VEL
LIN {X 0,Y 319.839,Z 644.646,A -85,B 0,C 180,E1 -15128.848,E2 -15128.848} C_VEL
LIN {X 0,Y 319.678,Z 644.666,A -85,B 0,C 180,E1 -15132.7,E2 -15132.7} C_VEL
LIN {X 0,Y 319.696,Z 644.664,A -85,B 0,C 180,E1 -15135.296,E2 -15135.296} C_VEL
LIN {X 0,Y 319.671,Z 644.665,A -85,B 0,C 180,E1 -15139.255,E2 -15139.255} C_VEL
LIN {X 0,Y 319.567,Z 644.678,A -85,B 0,C 180,E1 -15143.32,E2 -15143.32} C_VEL
LIN {X 0,Y 319.632,Z 644.669,A -85,B 0,C 180,E1 -15146.088,E2 -15146.088} C_VEL
LIN {X 0,Y 319.586,Z 644.675,A -85,B 0,C 180,E1 -15148.934,E2 -15148.934} C_VEL
LIN {X 0,Y 319.529,Z 644.684,A -85,B 0,C 180,E1 -15151.862,E2 -15151.862} C_VEL
LIN {X 0,Y 319.577,Z 644.676,A -85,B 0,C 180,E1 -15155.544,E2 -15155.544} C_VEL
LIN {X 0,Y 319.555,Z 644.679,A -85,B 0,C 180,E1 -15158.011,E2 -15158.011} C_VEL
LIN {X 0,Y 319.523,Z 644.683,A -85,B 0,C 180,E1 -15161.598,E2 -15161.598} C_VEL
LIN {X 0,Y 319.49,Z 644.69,A -85,B 0,C 180,E1 -15165.259,E2 -15165.259} C_VEL
LIN {X 0,Y 319.582,Z 644.881,A -85,B 0,C 180,E1 -15166.177,E2 -15166.177} C_VEL
LIN {X 0,Y 320.219,Z 648.208,A -85,B 0,C 180,E1 -15168.821,E2 -15168.821} C_VEL
LIN {X 0,Y 320.904,Z 652.653,A -85,B 0,C 180,E1 -15172.178,E2 -15172.178} C_VEL
LIN {X 0,Y 321.029,Z 655.322,A -85,B 0,C 180,E1 -15174.097,E2 -15174.097} C_VEL
LIN {X 0,Y 320.655,Z 659.208,A -85,B 0,C 180,E1 -15176.775,E2 -15176.775} C_VEL
LIN {X 0,Y 320.012,Z 664.623,A -85,B 0,C 180,E1 -15180.388,E2 -15180.388} C_VEL
LIN {X 0,Y 319.339,Z 670.889,A -85,B 0,C 180,E1 -15184.466,E2 -15184.466} C_VEL
LIN {X 0,Y 319.089,Z 674.215,A -85,B 0,C 180,E1 -15186.493,E2 -15186.493} C_VEL
LIN {X 0,Y 322.51,Z 687.976,A -85,B 0,C 180,E1 -15187.42,E2 -15187.42} C_VEL
LIN {X 0,Y 324.648,Z 700.171,A -85,B 0,C 180,E1 -15188.407,E2 -15188.407} C_VEL
LIN {X 0,Y 325.776,Z 713.07,A -85,B 0,C 180,E1 -15189.632,E2 -15189.632} C_VEL
LIN {X 0,Y 325.945,Z 719.37,A -85,B 0,C 180,E1 -15190.312,E2 -15190.312} C_VEL
LIN {X 0,Y 324.313,Z 730.978,A -85,B 0,C 180,E1 -15191.687,E2 -15191.687} C_VEL
LIN {X 0,Y 322.798,Z 741.542,A -85,B 0,C 180,E1 -15193.267,E2 -15193.267} C_VEL
LIN {X 0,Y 321.495,Z 749.791,A -85,B 0,C 180,E1 -15194.793,E2 -15194.793} C_VEL
LIN {X 0,Y 320.26,Z 758.03,A -85,B 0,C 180,E1 -15196.679,E2 -15196.679} C_VEL
LIN {X 0,Y 319.232,Z 764.706,A -85,B 0,C 180,E1 -15198.573,E2 -15198.573} C_VEL
LIN {X 0,Y 318.571,Z 770.044,A -85,B 0,C 180,E1 -15200.477,E2 -15200.477} C_VEL
LIN {X 0,Y 318.08,Z 774.198,A -85,B 0,C 180,E1 -15202.382,E2 -15202.382} C_VEL
LIN {X 0,Y 317.838,Z 778.442,A -85,B 0,C 180,E1 -15204.926,E2 -15204.926} C_VEL
LIN {X 0,Y 317.815,Z 780.062,A -85,B 0,C 180,E1 -15206.197,E2 -15206.197} C_VEL
LIN {X 0,Y 317.758,Z 781.271,A -85,B 0,C 180,E1 -15207.465,E2 -15207.465} C_VEL
LIN {X 0,Y 317.744,Z 782.034,A -85,B 0,C 180,E1 -15208.733,E2 -15208.733} C_VEL
LIN {X 0,Y 317.784,Z 782.385,A -85,B 0,C 180,E1 -15210.001,E2 -15210.001} C_VEL
LIN {X 0,Y 317.742,Z 782.341,A -85,B 0,C 180,E1 -15211.268,E2 -15211.268} C_VEL
LIN {X 0,Y 317.757,Z 781.906,A -85,B 0,C 180,E1 -15212.536,E2 -15212.536} C_VEL
LIN {X 0,Y 317.812,Z 781.04,A -85,B 0,C 180,E1 -15213.804,E2 -15213.804} C_VEL
LIN {X 0,Y 317.966,Z 778.063,A -85,B 0,C 180,E1 -15216.346,E2 -15216.346} C_VEL
LIN {X 0,Y 318.263,Z 774.684,A -85,B 0,C 180,E1 -15218.253,E2 -15218.253} C_VEL
LIN {X 0,Y 318.81,Z 770.238,A -85,B 0,C 180,E1 -15220.158,E2 -15220.158} C_VEL
LIN {X 0,Y 319.564,Z 764.607,A -85,B 0,C 180,E1 -15222.06,E2 -15222.06} C_VEL
LIN {X 0,Y 320.759,Z 757.618,A -85,B 0,C 180,E1 -15223.947,E2 -15223.947} C_VEL
LIN {X 0,Y 322.179,Z 748.938,A -85,B 0,C 180,E1 -15225.822,E2 -15225.822} C_VEL
LIN {X 0,Y 323.44,Z 740.092,A -85,B 0,C 180,E1 -15227.384,E2 -15227.384} C_VEL
LIN {X 0,Y 325.148,Z 729.286,A -85,B 0,C 180,E1 -15228.919,E2 -15228.919} C_VEL
LIN {X 0,Y 326.581,Z 718.501,A -85,B 0,C 180,E1 -15230.141,E2 -15230.141} C_VEL
LIN {X 0,Y 325.883,Z 706.779,A -85,B 0,C 180,E1 -15231.349,E2 -15231.349} C_VEL
LIN {X 0,Y 324.018,Z 694.262,A -85,B 0,C 180,E1 -15232.47,E2 -15232.47} C_VEL
LIN {X 0,Y 321.082,Z 681.614,A -85,B 0,C 180,E1 -15233.448,E2 -15233.448} C_VEL
LIN {X 0,Y 319.235,Z 675.041,A -85,B 0,C 180,E1 -15233.917,E2 -15233.917} C_VEL
LIN {X 0,Y 319.82,Z 669.714,A -85,B 0,C 180,E1 -15237.483,E2 -15237.483} C_VEL
LIN {X 0,Y 320.53,Z 664.358,A -85,B 0,C 180,E1 -15241.227,E2 -15241.227} C_VEL
LIN {X 0,Y 321.024,Z 660.976,A -85,B 0,C 180,E1 -15243.704,E2 -15243.704} C_VEL
LIN {X 0,Y 321.301,Z 657.752,A -85,B 0,C 180,E1 -15246.199,E2 -15246.199} C_VEL
LIN {X 0,Y 321.077,Z 653.95,A -85,B 0,C 180,E1 -15249.404,E2 -15249.404} C_VEL
LIN {X 0,Y 320.537,Z 650.296,A -85,B 0,C 180,E1 -15252.82,E2 -15252.82} C_VEL
LIN {X 0,Y 319.878,Z 646.322,A -85,B 0,C 180,E1 -15257.07,E2 -15257.07} C_VEL
LIN {X 0,Y 319.573,Z 644.959,A -85,B 0,C 180,E1 -15258.719,E2 -15258.719} C_VEL
LIN {X 0,Y 319.545,Z 644.684,A -85,B 0,C 180,E1 -15261.988,E2 -15261.988} C_VEL
LIN {X 0,Y 319.562,Z 644.681,A -85,B 0,C 180,E1 -15265.124,E2 -15265.124} C_VEL
LIN {X 0,Y 319.568,Z 644.679,A -85,B 0,C 180,E1 -15269.059,E2 -15269.059} C_VEL
LIN {X 0,Y 319.608,Z 644.675,A -85,B 0,C 180,E1 -15272.498,E2 -15272.498} C_VEL
LIN {X 0,Y 319.607,Z 644.674,A -85,B 0,C 180,E1 -15275.304,E2 -15275.304} C_VEL
LIN {X 0,Y 319.599,Z 644.676,A -85,B 0,C 180,E1 -15278.048,E2 -15278.048} C_VEL
LIN {X 0,Y 319.691,Z 644.665,A -85,B 0,C 180,E1 -15280.962,E2 -15280.962} C_VEL
LIN {X 0,Y 319.733,Z 644.659,A -85,B 0,C 180,E1 -15285.276,E2 -15285.276} C_VEL
LIN {X 0,Y 319.76,Z 644.652,A -85,B 0,C 180,E1 -15289.873,E2 -15289.873} C_VEL
LIN {X 0,Y 319.935,Z 644.631,A -85,B 0,C 180,E1 -15292.426,E2 -15292.426} C_VEL
LIN {X 0,Y 319.749,Z 644.658,A -85,B 0,C 180,E1 -15294.956,E2 -15294.956} C_VEL
LIN {X 0,Y 319.992,Z 644.625,A -85,B 0,C 180,E1 -15297.482,E2 -15297.482} C_VEL
LIN {X 0,Y 320.153,Z 644.607,A -85,B 0,C 180,E1 -15300,E2 -15300} C_VEL
LIN {X 0,Y 319.994,Z 644.629,A -85,B 0,C 180,E1 -15302.518,E2 -15302.518} C_VEL
LIN {X 0,Y 319.988,Z 646.061,A -85,B 0,C 180,E1 -15305.04,E2 -15305.04} C_VEL
LIN {X 0,Y 320.313,Z 647.932,A -85,B 0,C 180,E1 -15307.565,E2 -15307.565} C_VEL
LIN {X 0,Y 320.145,Z 650.046,A -85,B 0,C 180,E1 -15310.115,E2 -15310.115} C_VEL
LIN {X 0,Y 319.713,Z 653.466,A -85,B 0,C 180,E1 -15313.993,E2 -15313.993} C_VEL
LIN {X 0,Y 319.266,Z 657.201,A -85,B 0,C 180,E1 -15317.95,E2 -15317.95} C_VEL
LIN {X 0,Y 318.944,Z 660.341,A -85,B 0,C 180,E1 -15321.151,E2 -15321.151} C_VEL
LIN {X 0,Y 321.997,Z 669.291,A -85,B 0,C 180,E1 -15321.876,E2 -15321.876} C_VEL
LIN {X 0,Y 325.23,Z 680.678,A -85,B 0,C 180,E1 -15322.89,E2 -15322.89} C_VEL
LIN {X 0,Y 327.338,Z 691.367,A -85,B 0,C 180,E1 -15323.949,E2 -15323.949} C_VEL
LIN {X 0,Y 327.973,Z 697.417,A -85,B 0,C 180,E1 -15324.587,E2 -15324.587} C_VEL
LIN {X 0,Y 326.607,Z 707.674,A -85,B 0,C 180,E1 -15325.662,E2 -15325.662} C_VEL
LIN {X 0,Y 325.173,Z 717.828,A -85,B 0,C 180,E1 -15326.993,E2 -15326.993} C_VEL
LIN {X 0,Y 323.576,Z 727.462,A -85,B 0,C 180,E1 -15328.544,E2 -15328.544} C_VEL
LIN {X 0,Y 322.249,Z 735.356,A -85,B 0,C 180,E1 -15330.107,E2 -15330.107} C_VEL
LIN {X 0,Y 320.94,Z 743.383,A -85,B 0,C 180,E1 -15332.075,E2 -15332.075} C_VEL
LIN {X 0,Y 319.75,Z 749.95,A -85,B 0,C 180,E1 -15334.121,E2 -15334.121} C_VEL
LIN {X 0,Y 319.021,Z 754.545,A -85,B 0,C 180,E1 -15335.937,E2 -15335.937} C_VEL
LIN {X 0,Y 318.403,Z 758.811,A -85,B 0,C 180,E1 -15338.173,E2 -15338.173} C_VEL
LIN {X 0,Y 318.036,Z 761.09,A -85,B 0,C 180,E1 -15339.855,E2 -15339.855} C_VEL
LIN {X 0,Y 317.769,Z 762.674,A -85,B 0,C 180,E1 -15341.568,E2 -15341.568} C_VEL
LIN {X 0,Y 317.628,Z 763.51,A -85,B 0,C 180,E1 -15343.308,E2 -15343.308} C_VEL
LIN {X 0,Y 317.554,Z 763.572,A -85,B 0,C 180,E1 -15345.09,E2 -15345.09} C_VEL
LIN {X 0,Y 317.594,Z 762.835,A -85,B 0,C 180,E1 -15346.908,E2 -15346.908} C_VEL
LIN {X 0,Y 317.776,Z 761.233,A -85,B 0,C 180,E1 -15348.76,E2 -15348.76} C_VEL
LIN {X 0,Y 318.169,Z 757.674,A -85,B 0,C 180,E1 -15351.234,E2 -15351.234} C_VEL
LIN {X 0,Y 318.637,Z 753.009,A -85,B 0,C 180,E1 -15353.45,E2 -15353.45} C_VEL
LIN {X 0,Y 319.257,Z 747.34,A -85,B 0,C 180,E1 -15355.469,E2 -15355.469} C_VEL
LIN {X 0,Y 320.205,Z 740.197,A -85,B 0,C 180,E1 -15357.47,E2 -15357.47} C_VEL
LIN {X 0,Y 321.347,Z 731.343,A -85,B 0,C 180,E1 -15359.436,E2 -15359.436} C_VEL
LIN {X 0,Y 322.531,Z 722.213,A -85,B 0,C 180,E1 -15361.057,E2 -15361.057} C_VEL
LIN {X 0,Y 323.752,Z 712.148,A -85,B 0,C 180,E1 -15362.51,E2 -15362.51} C_VEL
LIN {X 0,Y 324.977,Z 700.46,A -85,B 0,C 180,E1 -15363.855,E2 -15363.855} C_VEL
LIN {X 0,Y 325.519,Z 692.733,A -85,B 0,C 180,E1 -15364.589,E2 -15364.589} C_VEL
LIN {X 0,Y 323.575,Z 681.187,A -85,B 0,C 180,E1 -15365.626,E2 -15365.626} C_VEL
LIN {X 0,Y 320.75,Z 668.25,A -85,B 0,C 180,E1 -15366.557,E2 -15366.557} C_VEL
LIN {X 0,Y 318.462,Z 658.991,A -85,B 0,C 180,E1 -15367.11,E2 -15367.11} C_VEL
LIN {X 0,Y 318.72,Z 655.043,A -85,B 0,C 180,E1 -15370.685,E2 -15370.685} C_VEL
LIN {X 0,Y 319.071,Z 650.731,A -85,B 0,C 180,E1 -15374.673,E2 -15374.673} C_VEL
LIN {X 0,Y 319.312,Z 647.962,A -85,B 0,C 180,E1 -15377.285,E2 -15377.285} C_VEL
LIN {X 0,Y 319.617,Z 644.674,A -85,B 0,C 180,E1 -15380.507,E2 -15380.507} C_VEL
LIN {X 0,Y 319.892,Z 644.636,A -85,B 0,C 180,E1 -15382.425,E2 -15382.425} C_VEL
LIN {X 0,Y 319.747,Z 644.658,A -85,B 0,C 180,E1 -15384.956,E2 -15384.956} C_VEL
LIN {X 0,Y 319.994,Z 644.622,A -85,B 0,C 180,E1 -15387.482,E2 -15387.482} C_VEL
LIN {X 0,Y 320.154,Z 644.602,A -85,B 0,C 180,E1 -15389.999,E2 -15389.999} C_VEL
LIN {X 0,Y 319.994,Z 644.624,A -85,B 0,C 180,E1 -15392.517,E2 -15392.517} C_VEL
LIN {X 0,Y 319.901,Z 644.635,A -85,B 0,C 180,E1 -15396.306,E2 -15396.306} C_VEL
LIN {X 0,Y 319.633,Z 644.672,A -85,B 0,C 180,E1 -15398.853,E2 -15398.853} C_VEL
LIN {X 0,Y 319.058,Z 644.896,A -85,B 0,C 180,E1 -15402.401,E2 -15402.401} C_VEL
LIN {X 0,Y 318.635,Z 650.662,A -85,B 0,C 180,E1 -15406.662,E2 -15406.662} C_VEL
LIN {X 0,Y 318.474,Z 654.27,A -85,B 0,C 180,E1 -15409.33,E2 -15409.33} C_VEL
LIN {X 0,Y 318.348,Z 657.899,A -85,B 0,C 180,E1 -15412.016,E2 -15412.016} C_VEL
LIN {X 0,Y 321.762,Z 672.25,A -85,B 0,C 180,E1 -15412.87,E2 -15412.87} C_VEL
LIN {X 0,Y 324.181,Z 684.472,A -85,B 0,C 180,E1 -15413.814,E2 -15413.814} C_VEL
LIN {X 0,Y 325.561,Z 693.531,A -85,B 0,C 180,E1 -15414.647,E2 -15414.647} C_VEL
LIN {X 0,Y 324.376,Z 705.517,A -85,B 0,C 180,E1 -15415.85,E2 -15415.85} C_VEL
LIN {X 0,Y 323.146,Z 716.02,A -85,B 0,C 180,E1 -15417.175,E2 -15417.175} C_VEL
LIN {X 0,Y 321.941,Z 725.743,A -85,B 0,C 180,E1 -15418.702,E2 -15418.702} C_VEL
LIN {X 0,Y 320.756,Z 734.871,A -85,B 0,C 180,E1 -15420.477,E2 -15420.477} C_VEL
LIN {X 0,Y 319.881,Z 741.919,A -85,B 0,C 180,E1 -15422.166,E2 -15422.166} C_VEL
LIN {X 0,Y 319.045,Z 748.663,A -85,B 0,C 180,E1 -15424.174,E2 -15424.174} C_VEL
LIN {X 0,Y 318.524,Z 753.28,A -85,B 0,C 180,E1 -15425.904,E2 -15425.904} C_VEL
LIN {X 0,Y 318.006,Z 757.946,A -85,B 0,C 180,E1 -15428.228,E2 -15428.228} C_VEL
LIN {X 0,Y 317.707,Z 760.376,A -85,B 0,C 180,E1 -15429.903,E2 -15429.903} C_VEL
LIN {X 0,Y 317.541,Z 762.086,A -85,B 0,C 180,E1 -15431.603,E2 -15431.603} C_VEL
LIN {X 0,Y 317.492,Z 763.031,A -85,B 0,C 180,E1 -15433.33,E2 -15433.33} C_VEL
LIN {X 0,Y 317.528,Z 763.236,A -85,B 0,C 180,E1 -15435.093,E2 -15435.093} C_VEL
LIN {X 0,Y 317.667,Z 762.657,A -85,B 0,C 180,E1 -15436.892,E2 -15436.892} C_VEL
LIN {X 0,Y 317.857,Z 761.221,A -85,B 0,C 180,E1 -15438.742,E2 -15438.742} C_VEL
LIN {X 0,Y 318.408,Z 757.841,A -85,B 0,C 180,E1 -15441.238,E2 -15441.238} C_VEL
LIN {X 0,Y 319.132,Z 753.245,A -85,B 0,C 180,E1 -15443.516,E2 -15443.516} C_VEL
LIN {X 0,Y 319.96,Z 747.866,A -85,B 0,C 180,E1 -15445.499,E2 -15445.499} C_VEL
LIN {X 0,Y 320.176,Z 746.739,A -85,B 0,C 180,E1 -15445.86,E2 -15445.86} C_VEL
LIN {X 0,Y 320.033,Z 743.8,A -85,B 0,C 180,E1 -15446.775,E2 -15446.775} C_VEL
LIN {X 0,Y 318.176,Z 738.764,A -85,B 0,C 180,E1 -15448.279,E2 -15448.279} C_VEL
LIN {X 0,Y 316.433,Z 733.207,A -85,B 0,C 180,E1 -15449.726,E2 -15449.726} C_VEL
LIN {X 0,Y 316.453,Z 729.342,A -85,B 0,C 180,E1 -15450.533,E2 -15450.533} C_VEL
LIN {X 0,Y 317.991,Z 720.055,A -85,B 0,C 180,E1 -15452.133,E2 -15452.133} C_VEL
LIN {X 0,Y 319.534,Z 709.886,A -85,B 0,C 180,E1 -15453.552,E2 -15453.552} C_VEL
LIN {X 0,Y 321.105,Z 698.373,A -85,B 0,C 180,E1 -15454.831,E2 -15454.831} C_VEL
LIN {X 0,Y 320.734,Z 693.194,A -85,B 0,C 180,E1 -15455.397,E2 -15455.397} C_VEL
LIN {X 0,Y 318.778,Z 682.147,A -85,B 0,C 180,E1 -15456.533,E2 -15456.533} C_VEL
LIN {X 0,Y 315.896,Z 671.087,A -85,B 0,C 180,E1 -15457.547,E2 -15457.547} C_VEL
LIN {X 0,Y 311.816,Z 658.948,A -85,B 0,C 180,E1 -15458.558,E2 -15458.558} C_VEL
LIN {X 0,Y 312.065,Z 654.926,A -85,B 0,C 180,E1 -15461.621,E2 -15461.621} C_VEL
LIN {X 0,Y 312.451,Z 649.599,A -85,B 0,C 180,E1 -15465.675,E2 -15465.675} C_VEL
LIN {X 0,Y 312.505,Z 645.734,A -85,B 0,C 180,E1 -15468.651,E2 -15468.651} C_VEL
LIN {X 0,Y 312.834,Z 645.522,A -85,B 0,C 180,E1 -15472.253,E2 -15472.253} C_VEL
LIN {X 0,Y 312.896,Z 645.514,A -85,B 0,C 180,E1 -15473.552,E2 -15473.552} C_VEL
LIN {X 0,Y 312.935,Z 645.505,A -85,B 0,C 180,E1 -15477.426,E2 -15477.426} C_VEL
LIN {X 0,Y 313.118,Z 645.484,A -85,B 0,C 180,E1 -15480,E2 -15480} C_VEL
LIN {X 0,Y 312.935,Z 645.507,A -85,B 0,C 180,E1 -15482.574,E2 -15482.574} C_VEL
LIN {X 0,Y 312.907,Z 645.51,A -85,B 0,C 180,E1 -15486.448,E2 -15486.448} C_VEL
LIN {X 0,Y 312.784,Z 645.525,A -85,B 0,C 180,E1 -15489.049,E2 -15489.049} C_VEL
LIN {X 0,Y 312.631,Z 645.544,A -85,B 0,C 180,E1 -15492.991,E2 -15492.991} C_VEL
LIN {X 0,Y 312.634,Z 645.544,A -85,B 0,C 180,E1 -15495.65,E2 -15495.65} C_VEL
LIN {X 0,Y 312.627,Z 645.542,A -85,B 0,C 180,E1 -15499.237,E2 -15499.237} C_VEL
LIN {X 0,Y 312.542,Z 645.555,A -85,B 0,C 180,E1 -15502.79,E2 -15502.79} C_VEL
LIN {X 0,Y 312.599,Z 645.545,A -85,B 0,C 180,E1 -15505.936,E2 -15505.936} C_VEL
LIN {X 0,Y 312.542,Z 645.555,A -85,B 0,C 180,E1 -15509.65,E2 -15509.65} C_VEL
LIN {X 0,Y 312.516,Z 645.556,A -85,B 0,C 180,E1 -15513.689,E2 -15513.689} C_VEL
LIN {X 0,Y 312.523,Z 645.555,A -85,B 0,C 180,E1 -15517.386,E2 -15517.386} C_VEL
LIN {X 0,Y 312.487,Z 645.562,A -85,B 0,C 180,E1 -15520.71,E2 -15520.71} C_VEL
LIN {X 0,Y 312.45,Z 645.567,A -85,B 0,C 180,E1 -15524.21,E2 -15524.21} C_VEL
LIN {X 0,Y 312.5,Z 645.594,A -85,B 0,C 180,E1 -15525.8,E2 -15525.8} C_VEL
LIN {X 0,Y 313.316,Z 650.088,A -85,B 0,C 180,E1 -15529.422,E2 -15529.422} C_VEL
LIN {X 0,Y 313.829,Z 652.92,A -85,B 0,C 180,E1 -15531.61,E2 -15531.61} C_VEL
LIN {X 0,Y 313.948,Z 656.729,A -85,B 0,C 180,E1 -15534.407,E2 -15534.407} C_VEL
LIN {X 0,Y 313.45,Z 661.057,A -85,B 0,C 180,E1 -15537.445,E2 -15537.445} C_VEL
LIN {X 0,Y 312.807,Z 666.576,A -85,B 0,C 180,E1 -15541.192,E2 -15541.192} C_VEL
LIN {X 0,Y 312.123,Z 672.895,A -85,B 0,C 180,E1 -15545.383,E2 -15545.383} C_VEL
LIN {X 0,Y 312.064,Z 673.471,A -85,B 0,C 180,E1 -15545.76,E2 -15545.76} C_VEL
LIN {X 0,Y 313.66,Z 679.698,A -85,B 0,C 180,E1 -15546.185,E2 -15546.185} C_VEL
LIN {X 0,Y 316.659,Z 692.397,A -85,B 0,C 180,E1 -15547.168,E2 -15547.168} C_VEL
LIN {X 0,Y 318.352,Z 703.865,A -85,B 0,C 180,E1 -15548.177,E2 -15548.177} C_VEL
LIN {X 0,Y 319.178,Z 715.465,A -85,B 0,C 180,E1 -15549.372,E2 -15549.372} C_VEL
LIN {X 0,Y 319.123,Z 721.284,A -85,B 0,C 180,E1 -15550.041,E2 -15550.041} C_VEL
LIN {X 0,Y 317.419,Z 732.485,A -85,B 0,C 180,E1 -15551.442,E2 -15551.442} C_VEL
LIN {X 0,Y 316.044,Z 741.597,A -85,B 0,C 180,E1 -15552.864,E2 -15552.864} C_VEL
LIN {X 0,Y 314.643,Z 749.944,A -85,B 0,C 180,E1 -15554.453,E2 -15554.453} C_VEL
LIN {X 0,Y 313.349,Z 758.124,A -85,B 0,C 180,E1 -15556.38,E2 -15556.38} C_VEL
LIN {X 0,Y 312.238,Z 764.74,A -85,B 0,C 180,E1 -15558.313,E2 -15558.313} C_VEL
LIN {X 0,Y 311.534,Z 770.02,A -85,B 0,C 180,E1 -15560.26,E2 -15560.26} C_VEL
LIN {X 0,Y 311.022,Z 774.122,A -85,B 0,C 180,E1 -15562.209,E2 -15562.209} C_VEL
LIN {X 0,Y 310.757,Z 778.131,A -85,B 0,C 180,E1 -15564.81,E2 -15564.81} C_VEL
LIN {X 0,Y 310.727,Z 779.766,A -85,B 0,C 180,E1 -15566.11,E2 -15566.11} C_VEL
LIN {X 0,Y 310.682,Z 780.995,A -85,B 0,C 180,E1 -15567.407,E2 -15567.407} C_VEL
LIN {X 0,Y 310.658,Z 781.794,A -85,B 0,C 180,E1 -15568.704,E2 -15568.704} C_VEL
LIN {X 0,Y 310.694,Z 782.163,A -85,B 0,C 180,E1 -15570.001,E2 -15570.001} C_VEL
LIN {X 0,Y 310.656,Z 782.136,A -85,B 0,C 180,E1 -15571.297,E2 -15571.297} C_VEL
LIN {X 0,Y 310.681,Z 781.718,A -85,B 0,C 180,E1 -15572.594,E2 -15572.594} C_VEL
LIN {X 0,Y 310.724,Z 780.886,A -85,B 0,C 180,E1 -15573.891,E2 -15573.891} C_VEL
LIN {X 0,Y 310.897,Z 777.942,A -85,B 0,C 180,E1 -15576.49,E2 -15576.49} C_VEL
LIN {X 0,Y 311.22,Z 774.598,A -85,B 0,C 180,E1 -15578.441,E2 -15578.441} C_VEL
LIN {X 0,Y 311.798,Z 770.202,A -85,B 0,C 180,E1 -15580.389,E2 -15580.389} C_VEL
LIN {X 0,Y 312.794,Z 763.602,A -85,B 0,C 180,E1 -15582.655,E2 -15582.655} C_VEL
LIN {X 0,Y 314.112,Z 756.392,A -85,B 0,C 180,E1 -15584.579,E2 -15584.579} C_VEL
LIN {X 0,Y 315.449,Z 748.263,A -85,B 0,C 180,E1 -15586.345,E2 -15586.345} C_VEL
LIN {X 0,Y 317.013,Z 738.414,A -85,B 0,C 180,E1 -15588.082,E2 -15588.082} C_VEL
LIN {X 0,Y 318.668,Z 728.444,A -85,B 0,C 180,E1 -15589.486,E2 -15589.486} C_VEL
LIN {X 0,Y 319.89,Z 719.061,A -85,B 0,C 180,E1 -15590.581,E2 -15590.581} C_VEL
LIN {X 0,Y 319.279,Z 707.754,A -85,B 0,C 180,E1 -15591.804,E2 -15591.804} C_VEL
LIN {X 0,Y 317.534,Z 695.561,A -85,B 0,C 180,E1 -15592.954,E2 -15592.954} C_VEL
LIN {X 0,Y 314.888,Z 684.077,A -85,B 0,C 180,E1 -15593.91,E2 -15593.91} C_VEL
LIN {X 0,Y 312.284,Z 674.804,A -85,B 0,C 180,E1 -15594.604,E2 -15594.604} C_VEL
LIN {X 0,Y 313.049,Z 668.64,A -85,B 0,C 180,E1 -15598.889,E2 -15598.889} C_VEL
LIN {X 0,Y 313.742,Z 663.677,A -85,B 0,C 180,E1 -15602.522,E2 -15602.522} C_VEL
LIN {X 0,Y 314.228,Z 659.766,A -85,B 0,C 180,E1 -15605.558,E2 -15605.558} C_VEL
LIN {X 0,Y 314.194,Z 656.308,A -85,B 0,C 180,E1 -15608.474,E2 -15608.474} C_VEL
LIN {X 0,Y 313.693,Z 652.285,A -85,B 0,C 180,E1 -15612.231,E2 -15612.231} C_VEL
LIN {X 0,Y 313.07,Z 648.836,A -85,B 0,C 180,E1 -15615.919,E2 -15615.919} C_VEL
LIN {X 0,Y 312.515,Z 645.614,A -85,B 0,C 180,E1 -15619.873,E2 -15619.873} C_VEL
LIN {X 0,Y 312.537,Z 645.556,A -85,B 0,C 180,E1 -15624.05,E2 -15624.05} C_VEL
LIN {X 0,Y 312.505,Z 645.558,A -85,B 0,C 180,E1 -15627.334,E2 -15627.334} C_VEL
LIN {X 0,Y 312.546,Z 645.552,A -85,B 0,C 180,E1 -15631.279,E2 -15631.279} C_VEL
LIN {X 0,Y 312.587,Z 645.55,A -85,B 0,C 180,E1 -15634.711,E2 -15634.711} C_VEL
LIN {X 0,Y 312.589,Z 645.549,A -85,B 0,C 180,E1 -15637.529,E2 -15637.529} C_VEL
LIN {X 0,Y 312.64,Z 645.543,A -85,B 0,C 180,E1 -15641.656,E2 -15641.656} C_VEL
LIN {X 0,Y 312.696,Z 645.536,A -85,B 0,C 180,E1 -15645.686,E2 -15645.686} C_VEL
LIN {X 0,Y 312.704,Z 645.532,A -85,B 0,C 180,E1 -15649.642,E2 -15649.642} C_VEL
LIN {X 0,Y 312.874,Z 645.51,A -85,B 0,C 180,E1 -15652.254,E2 -15652.254} C_VEL
LIN {X 0,Y 312.72,Z 645.533,A -85,B 0,C 180,E1 -15654.842,E2 -15654.842} C_VEL
LIN {X 0,Y 312.992,Z 645.498,A -85,B 0,C 180,E1 -15658.713,E2 -15658.713} C_VEL
LIN {X 0,Y 312.993,Z 645.5,A -85,B 0,C 180,E1 -15661.287,E2 -15661.287} C_VEL
LIN {X 0,Y 312.973,Z 645.665,A -85,B 0,C 180,E1 -15662.574,E2 -15662.574} C_VEL
LIN {X 0,Y 313.228,Z 648.646,A -85,B 0,C 180,E1 -15666.83,E2 -15666.83} C_VEL
LIN {X 0,Y 313.276,Z 650.486,A -85,B 0,C 180,E1 -15669.214,E2 -15669.214} C_VEL
LIN {X 0,Y 312.8,Z 653.69,A -85,B 0,C 180,E1 -15672.984,E2 -15672.984} C_VEL
LIN {X 0,Y 312.461,Z 656.093,A -85,B 0,C 180,E1 -15675.659,E2 -15675.659} C_VEL
LIN {X 0,Y 312.037,Z 659.933,A -85,B 0,C 180,E1 -15679.746,E2 -15679.746} C_VEL
LIN {X 0,Y 311.975,Z 660.605,A -85,B 0,C 180,E1 -15680.437,E2 -15680.437} C_VEL
LIN {X 0,Y 312.996,Z 663.772,A -85,B 0,C 180,E1 -15680.711,E2 -15680.711} C_VEL
LIN {X 0,Y 317.05,Z 675.914,A -85,B 0,C 180,E1 -15681.796,E2 -15681.796} C_VEL
LIN {X 0,Y 319.913,Z 687.59,A -85,B 0,C 180,E1 -15682.951,E2 -15682.951} C_VEL
LIN {X 0,Y 321.381,Z 697.451,A -85,B 0,C 180,E1 -15684.035,E2 -15684.035} C_VEL
LIN {X 0,Y 319.906,Z 708.945,A -85,B 0,C 180,E1 -15685.293,E2 -15685.293} C_VEL
LIN {X 0,Y 318.32,Z 719.475,A -85,B 0,C 180,E1 -15686.734,E2 -15686.734} C_VEL
LIN {X 0,Y 316.697,Z 728.865,A -85,B 0,C 180,E1 -15688.317,E2 -15688.317} C_VEL
LIN {X 0,Y 315.071,Z 737.949,A -85,B 0,C 180,E1 -15690.243,E2 -15690.243} C_VEL
LIN {X 0,Y 313.849,Z 744.921,A -85,B 0,C 180,E1 -15692.088,E2 -15692.088} C_VEL
LIN {X 0,Y 312.642,Z 751.276,A -85,B 0,C 180,E1 -15694.193,E2 -15694.193} C_VEL
LIN {X 0,Y 311.69,Z 756.881,A -85,B 0,C 180,E1 -15696.693,E2 -15696.693} C_VEL
LIN {X 0,Y 311.068,Z 760.842,A -85,B 0,C 180,E1 -15699.243,E2 -15699.243} C_VEL
LIN {X 0,Y 310.67,Z 763.064,A -85,B 0,C 180,E1 -15701.709,E2 -15701.709} C_VEL
LIN {X 0,Y 310.505,Z 763.802,A -85,B 0,C 180,E1 -15703.59,E2 -15703.59} C_VEL
LIN {X 0,Y 310.45,Z 763.719,A -85,B 0,C 180,E1 -15705.43,E2 -15705.43} C_VEL
LIN {X 0,Y 310.534,Z 762.816,A -85,B 0,C 180,E1 -15707.237,E2 -15707.237} C_VEL
LIN {X 0,Y 310.701,Z 761.175,A -85,B 0,C 180,E1 -15709.006,E2 -15709.006} C_VEL
LIN {X 0,Y 310.992,Z 758.81,A -85,B 0,C 180,E1 -15710.745,E2 -15710.745} C_VEL
LIN {X 0,Y 311.279,Z 755.733,A -85,B 0,C 180,E1 -15712.439,E2 -15712.439} C_VEL
LIN {X 0,Y 311.897,Z 750.491,A -85,B 0,C 180,E1 -15714.621,E2 -15714.621} C_VEL
LIN {X 0,Y 312.782,Z 743.462,A -85,B 0,C 180,E1 -15716.857,E2 -15716.857} C_VEL
LIN {X 0,Y 313.783,Z 736.136,A -85,B 0,C 180,E1 -15718.704,E2 -15718.704} C_VEL
LIN {X 0,Y 314.997,Z 726.712,A -85,B 0,C 180,E1 -15720.603,E2 -15720.603} C_VEL
LIN {X 0,Y 316.317,Z 716.926,A -85,B 0,C 180,E1 -15722.187,E2 -15722.187} C_VEL
LIN {X 0,Y 317.565,Z 706.508,A -85,B 0,C 180,E1 -15723.552,E2 -15723.552} C_VEL
LIN {X 0,Y 318.698,Z 695.406,A -85,B 0,C 180,E1 -15724.708,E2 -15724.708} C_VEL
LIN {X 0,Y 317.376,Z 685.736,A -85,B 0,C 180,E1 -15725.642,E2 -15725.642} C_VEL
LIN {X 0,Y 314.749,Z 672.761,A -85,B 0,C 180,E1 -15726.685,E2 -15726.685} C_VEL
LIN {X 0,Y 311.418,Z 659.205,A -85,B 0,C 180,E1 -15727.538,E2 -15727.538} C_VEL
LIN {X 0,Y 311.743,Z 654.8,A -85,B 0,C 180,E1 -15731.601,E2 -15731.601} C_VEL
LIN {X 0,Y 312.138,Z 650.518,A -85,B 0,C 180,E1 -15735.66,E2 -15735.66} C_VEL
LIN {X 0,Y 312.48,Z 646.449,A -85,B 0,C 180,E1 -15739.634,E2 -15739.634} C_VEL
LIN {X 0,Y 312.611,Z 645.547,A -85,B 0,C 180,E1 -15740.619,E2 -15740.619} C_VEL
LIN {X 0,Y 312.895,Z 645.507,A -85,B 0,C 180,E1 -15743.551,E2 -15743.551} C_VEL
LIN {X 0,Y 312.94,Z 645.501,A -85,B 0,C 180,E1 -15747.425,E2 -15747.425} C_VEL
LIN {X 0,Y 313.106,Z 645.48,A -85,B 0,C 180,E1 -15749.999,E2 -15749.999} C_VEL
LIN {X 0,Y 312.94,Z 645.503,A -85,B 0,C 180,E1 -15752.574,E2 -15752.574} C_VEL
LIN {X 0,Y 312.837,Z 645.516,A -85,B 0,C 180,E1 -15756.449,E2 -15756.449} C_VEL
LIN {X 0,Y 312.557,Z 645.552,A -85,B 0,C 180,E1 -15759.055,E2 -15759.055} C_VEL
LIN {X 0,Y 312.012,Z 645.735,A -85,B 0,C 180,E1 -15762.355,E2 -15762.355} C_VEL
LIN {X 0,Y 311.632,Z 650.188,A -85,B 0,C 180,E1 -15765.701,E2 -15765.701} C_VEL
LIN {X 0,Y 311.47,Z 654.072,A -85,B 0,C 180,E1 -15768.614,E2 -15768.614} C_VEL
LIN {X 0,Y 311.291,Z 658.063,A -85,B 0,C 180,E1 -15771.58,E2 -15771.58} C_VEL
LIN {X 0,Y 314.653,Z 672.035,A -85,B 0,C 180,E1 -15772.431,E2 -15772.431} C_VEL
LIN {X 0,Y 317.013,Z 683.811,A -85,B 0,C 180,E1 -15773.351,E2 -15773.351} C_VEL
LIN {X 0,Y 318.619,Z 693.389,A -85,B 0,C 180,E1 -15774.256,E2 -15774.256} C_VEL
LIN {X 0,Y 317.772,Z 703.329,A -85,B 0,C 180,E1 -15775.249,E2 -15775.249} C_VEL
LIN {X 0,Y 316.554,Z 713.854,A -85,B 0,C 180,E1 -15776.548,E2 -15776.548} C_VEL
LIN {X 0,Y 315.278,Z 723.96,A -85,B 0,C 180,E1 -15778.092,E2 -15778.092} C_VEL
LIN {X 0,Y 314.011,Z 733.318,A -85,B 0,C 180,E1 -15779.866,E2 -15779.866} C_VEL
LIN {X 0,Y 312.986,Z 741.026,A -85,B 0,C 180,E1 -15781.686,E2 -15781.686} C_VEL
LIN {X 0,Y 312.066,Z 748.463,A -85,B 0,C 180,E1 -15783.888,E2 -15783.888} C_VEL
LIN {X 0,Y 311.422,Z 753.767,A -85,B 0,C 180,E1 -15785.926,E2 -15785.926} C_VEL
LIN {X 0,Y 310.993,Z 757.412,A -85,B 0,C 180,E1 -15787.725,E2 -15787.725} C_VEL
LIN {X 0,Y 310.635,Z 760.384,A -85,B 0,C 180,E1 -15789.714,E2 -15789.714} C_VEL
LIN {X 0,Y 310.453,Z 762.318,A -85,B 0,C 180,E1 -15791.664,E2 -15791.664} C_VEL
LIN {X 0,Y 310.397,Z 763.303,A -85,B 0,C 180,E1 -15793.569,E2 -15793.569} C_VEL
LIN {X 0,Y 310.441,Z 763.414,A -85,B 0,C 180,E1 -15795.428,E2 -15795.428} C_VEL
LIN {X 0,Y 310.602,Z 762.729,A -85,B 0,C 180,E1 -15797.249,E2 -15797.249} C_VEL
LIN {X 0,Y 310.824,Z 761.306,A -85,B 0,C 180,E1 -15799.026,E2 -15799.026} C_VEL
LIN {X 0,Y 311.388,Z 757.995,A -85,B 0,C 180,E1 -15801.505,E2 -15801.505} C_VEL
LIN {X 0,Y 311.984,Z 754.464,A -85,B 0,C 180,E1 -15803.348,E2 -15803.348} C_VEL
LIN {X 0,Y 312.885,Z 749.224,A -85,B 0,C 180,E1 -15805.447,E2 -15805.447} C_VEL
LIN {X 0,Y 314.047,Z 742.536,A -85,B 0,C 180,E1 -15807.514,E2 -15807.514} C_VEL
LIN {X 0,Y 315.51,Z 734.707,A -85,B 0,C 180,E1 -15809.429,E2 -15809.429} C_VEL
LIN {X 0,Y 316.453,Z 729.342,A -85,B 0,C 180,E1 -15810.533,E2 -15810.533} C_VEL
LIN {X 0,Y 316.515,Z 725.32,A -85,B 0,C 180,E1 -15811.316,E2 -15811.316} C_VEL
LIN {X 0,Y 314.967,Z 718.605,A -85,B 0,C 180,E1 -15812.615,E2 -15812.615} C_VEL
LIN {X 0,Y 313.459,Z 711.496,A -85,B 0,C 180,E1 -15813.838,E2 -15813.838} C_VEL
LIN {X 0,Y 313.54,Z 706.761,A -85,B 0,C 180,E1 -15814.48,E2 -15814.48} C_VEL
LIN {X 0,Y 314.618,Z 698.265,A -85,B 0,C 180,E1 -15815.414,E2 -15815.414} C_VEL
LIN {X 0,Y 313.135,Z 687.667,A -85,B 0,C 180,E1 -15816.606,E2 -15816.606} C_VEL
LIN {X 0,Y 310.614,Z 676.658,A -85,B 0,C 180,E1 -15817.721,E2 -15817.721} C_VEL
LIN {X 0,Y 306.706,Z 664.569,A -85,B 0,C 180,E1 -15818.844,E2 -15818.844} C_VEL
LIN {X 0,Y 304.84,Z 659.174,A -85,B 0,C 180,E1 -15819.283,E2 -15819.283} C_VEL
LIN {X 0,Y 305.11,Z 654.927,A -85,B 0,C 180,E1 -15822.576,E2 -15822.576} C_VEL
LIN {X 0,Y 305.423,Z 651.355,A -85,B 0,C 180,E1 -15825.338,E2 -15825.338} C_VEL
LIN {X 0,Y 305.56,Z 647.884,A -85,B 0,C 180,E1 -15828.053,E2 -15828.053} C_VEL
LIN {X 0,Y 305.497,Z 646.433,A -85,B 0,C 180,E1 -15829.395,E2 -15829.395} C_VEL
LIN {X 0,Y 305.769,Z 646.401,A -85,B 0,C 180,E1 -15832.073,E2 -15832.073} C_VEL
LIN {X 0,Y 305.685,Z 646.411,A -85,B 0,C 180,E1 -15834.723,E2 -15834.723} C_VEL
LIN {X 0,Y 305.956,Z 646.374,A -85,B 0,C 180,E1 -15838.684,E2 -15838.684} C_VEL
LIN {X 0,Y 305.956,Z 646.377,A -85,B 0,C 180,E1 -15841.316,E2 -15841.316} C_VEL
LIN {X 0,Y 305.849,Z 646.39,A -85,B 0,C 180,E1 -15846.597,E2 -15846.597} C_VEL
LIN {X 0,Y 305.732,Z 646.402,A -85,B 0,C 180,E1 -15849.26,E2 -15849.26} C_VEL
LIN {X 0,Y 305.586,Z 646.422,A -85,B 0,C 180,E1 -15853.296,E2 -15853.296} C_VEL
LIN {X 0,Y 305.59,Z 646.419,A -85,B 0,C 180,E1 -15856.02,E2 -15856.02} C_VEL
LIN {X 0,Y 305.573,Z 646.421,A -85,B 0,C 180,E1 -15859.445,E2 -15859.445} C_VEL
LIN {X 0,Y 305.487,Z 646.433,A -85,B 0,C 180,E1 -15863.042,E2 -15863.042} C_VEL
LIN {X 0,Y 305.544,Z 646.423,A -85,B 0,C 180,E1 -15866.228,E2 -15866.228} C_VEL
LIN {X 0,Y 305.493,Z 646.431,A -85,B 0,C 180,E1 -15869.05,E2 -15869.05} C_VEL
LIN {X 0,Y 305.441,Z 646.439,A -85,B 0,C 180,E1 -15871.953,E2 -15871.953} C_VEL
LIN {X 0,Y 305.459,Z 646.435,A -85,B 0,C 180,E1 -15875.114,E2 -15875.114} C_VEL
LIN {X 0,Y 305.447,Z 646.439,A -85,B 0,C 180,E1 -15878.529,E2 -15878.529} C_VEL
LIN {X 0,Y 305.452,Z 646.437,A -85,B 0,C 180,E1 -15882.586,E2 -15882.586} C_VEL
LIN {X 0,Y 305.468,Z 646.553,A -85,B 0,C 180,E1 -15885.612,E2 -15885.612} C_VEL
LIN {X 0,Y 306.261,Z 650.919,A -85,B 0,C 180,E1 -15889.225,E2 -15889.225} C_VEL
LIN {X 0,Y 306.821,Z 654.179,A -85,B 0,C 180,E1 -15891.797,E2 -15891.797} C_VEL
LIN {X 0,Y 306.934,Z 657.478,A -85,B 0,C 180,E1 -15894.277,E2 -15894.277} C_VEL
LIN {X 0,Y 306.403,Z 661.814,A -85,B 0,C 180,E1 -15897.385,E2 -15897.385} C_VEL
LIN {X 0,Y 305.741,Z 667.214,A -85,B 0,C 180,E1 -15901.137,E2 -15901.137} C_VEL
LIN {X 0,Y 305.08,Z 672.941,A -85,B 0,C 180,E1 -15905.025,E2 -15905.025} C_VEL
LIN {X 0,Y 306.065,Z 676.59,A -85,B 0,C 180,E1 -15905.274,E2 -15905.274} C_VEL
LIN {X 0,Y 309.366,Z 689.575,A -85,B 0,C 180,E1 -15906.293,E2 -15906.293} C_VEL
LIN {X 0,Y 311.519,Z 702.298,A -85,B 0,C 180,E1 -15907.448,E2 -15907.448} C_VEL
LIN {X 0,Y 312.445,Z 714.583,A -85,B 0,C 180,E1 -15908.726,E2 -15908.726} C_VEL
LIN {X 0,Y 312.481,Z 721.876,A -85,B 0,C 180,E1 -15909.598,E2 -15909.598} C_VEL
LIN {X 0,Y 310.729,Z 732.919,A -85,B 0,C 180,E1 -15911.027,E2 -15911.027} C_VEL
LIN {X 0,Y 309.279,Z 741.872,A -85,B 0,C 180,E1 -15912.478,E2 -15912.478} C_VEL
LIN {X 0,Y 307.804,Z 750.115,A -85,B 0,C 180,E1 -15914.099,E2 -15914.099} C_VEL
LIN {X 0,Y 306.445,Z 758.218,A -85,B 0,C 180,E1 -15916.067,E2 -15916.067} C_VEL
LIN {X 0,Y 305.249,Z 764.783,A -85,B 0,C 180,E1 -15918.041,E2 -15918.041} C_VEL
LIN {X 0,Y 304.502,Z 770.01,A -85,B 0,C 180,E1 -15920.032,E2 -15920.032} C_VEL
LIN {X 0,Y 303.986,Z 774.066,A -85,B 0,C 180,E1 -15922.027,E2 -15922.027} C_VEL
LIN {X 0,Y 303.686,Z 777.858,A -85,B 0,C 180,E1 -15924.689,E2 -15924.689} C_VEL
LIN {X 0,Y 303.608,Z 780.718,A -85,B 0,C 180,E1 -15927.347,E2 -15927.347} C_VEL
LIN {X 0,Y 303.575,Z 781.552,A -85,B 0,C 180,E1 -15928.674,E2 -15928.674} C_VEL
LIN {X 0,Y 303.606,Z 781.94,A -85,B 0,C 180,E1 -15930.001,E2 -15930.001} C_VEL
LIN {X 0,Y 303.573,Z 781.931,A -85,B 0,C 180,E1 -15931.327,E2 -15931.327} C_VEL
LIN {X 0,Y 303.606,Z 781.531,A -85,B 0,C 180,E1 -15932.654,E2 -15932.654} C_VEL
LIN {X 0,Y 303.639,Z 780.732,A -85,B 0,C 180,E1 -15933.982,E2 -15933.982} C_VEL
LIN {X 0,Y 303.696,Z 779.071,A -85,B 0,C 180,E1 -15935.679,E2 -15935.679} C_VEL
LIN {X 0,Y 304.025,Z 775.768,A -85,B 0,C 180,E1 -15937.973,E2 -15937.973} C_VEL
LIN {X 0,Y 304.527,Z 771.778,A -85,B 0,C 180,E1 -15939.968,E2 -15939.968} C_VEL
LIN {X 0,Y 305.48,Z 765.688,A -85,B 0,C 180,E1 -15942.288,E2 -15942.288} C_VEL
LIN {X 0,Y 306.767,Z 759.043,A -85,B 0,C 180,E1 -15944.258,E2 -15944.258} C_VEL
LIN {X 0,Y 308.256,Z 751.112,A -85,B 0,C 180,E1 -15946.155,E2 -15946.155} C_VEL
LIN {X 0,Y 309.622,Z 742.529,A -85,B 0,C 180,E1 -15947.844,E2 -15947.844} C_VEL
LIN {X 0,Y 311.407,Z 732.398,A -85,B 0,C 180,E1 -15949.444,E2 -15949.444} C_VEL
LIN {X 0,Y 313.213,Z 721.098,A -85,B 0,C 180,E1 -15950.868,E2 -15950.868} C_VEL
LIN {X 0,Y 312.852,Z 710.59,A -85,B 0,C 180,E1 -15952.082,E2 -15952.082} C_VEL
LIN {X 0,Y 311.355,Z 698.813,A -85,B 0,C 180,E1 -15953.284,E2 -15953.284} C_VEL
LIN {X 0,Y 308.771,Z 686.684,A -85,B 0,C 180,E1 -15954.378,E2 -15954.378} C_VEL
LIN {X 0,Y 305.423,Z 675.252,A -85,B 0,C 180,E1 -15955.304,E2 -15955.304} C_VEL
LIN {X 0,Y 305.342,Z 674.529,A -85,B 0,C 180,E1 -15955.374,E2 -15955.374} C_VEL
LIN {X 0,Y 306.068,Z 669.144,A -85,B 0,C 180,E1 -15959.242,E2 -15959.242} C_VEL
LIN {X 0,Y 306.864,Z 663.72,A -85,B 0,C 180,E1 -15963.344,E2 -15963.344} C_VEL
LIN {X 0,Y 307.304,Z 659.85,A -85,B 0,C 180,E1 -15966.486,E2 -15966.486} C_VEL
LIN {X 0,Y 307.156,Z 657.095,A -85,B 0,C 180,E1 -15968.927,E2 -15968.927} C_VEL
LIN {X 0,Y 306.799,Z 654.279,A -85,B 0,C 180,E1 -15971.63,E2 -15971.63} C_VEL
LIN {X 0,Y 306.211,Z 650.808,A -85,B 0,C 180,E1 -15975.357,E2 -15975.357} C_VEL
LIN {X 0,Y 305.784,Z 648.449,A -85,B 0,C 180,E1 -15978.201,E2 -15978.201} C_VEL
LIN {X 0,Y 305.582,Z 647.143,A -85,B 0,C 180,E1 -15979.912,E2 -15979.912} C_VEL
LIN {X 0,Y 305.469,Z 646.436,A -85,B 0,C 180,E1 -15981.596,E2 -15981.596} C_VEL
LIN {X 0,Y 305.464,Z 646.436,A -85,B 0,C 180,E1 -15984.887,E2 -15984.887} C_VEL
LIN {X 0,Y 305.451,Z 646.437,A -85,B 0,C 180,E1 -15988.356,E2 -15988.356} C_VEL
LIN {X 0,Y 305.515,Z 646.428,A -85,B 0,C 180,E1 -15991.113,E2 -15991.113} C_VEL
LIN {X 0,Y 305.567,Z 646.42,A -85,B 0,C 180,E1 -15994.087,E2 -15994.087} C_VEL
LIN {X 0,Y 305.502,Z 646.433,A -85,B 0,C 180,E1 -15998.403,E2 -15998.403} C_VEL
LIN {X 0,Y 305.592,Z 646.42,A -85,B 0,C 180,E1 -16001.218,E2 -16001.218} C_VEL
LIN {X 0,Y 305.651,Z 646.413,A -85,B 0,C 180,E1 -16005.349,E2 -16005.349} C_VEL
LIN {X 0,Y 305.641,Z 646.413,A -85,B 0,C 180,E1 -16009.4,E2 -16009.4} C_VEL
LIN {X 0,Y 305.815,Z 646.39,A -85,B 0,C 180,E1 -16012.074,E2 -16012.074} C_VEL
LIN {X 0,Y 305.691,Z 646.408,A -85,B 0,C 180,E1 -16014.724,E2 -16014.724} C_VEL
LIN {X 0,Y 305.959,Z 646.374,A -85,B 0,C 180,E1 -16018.684,E2 -16018.684} C_VEL
LIN {X 0,Y 305.961,Z 646.376,A -85,B 0,C 180,E1 -16021.316,E2 -16021.316} C_VEL
LIN {X 0,Y 305.921,Z 647.958,A -85,B 0,C 180,E1 -16023.952,E2 -16023.952} C_VEL
LIN {X 0,Y 306.237,Z 649.925,A -85,B 0,C 180,E1 -16026.837,E2 -16026.837} C_VEL
LIN {X 0,Y 306.25,Z 651.801,A -85,B 0,C 180,E1 -16029.322,E2 -16029.322} C_VEL
LIN {X 0,Y 305.734,Z 655.09,A -85,B 0,C 180,E1 -16033.29,E2 -16033.29} C_VEL
LIN {X 0,Y 305.39,Z 657.51,A -85,B 0,C 180,E1 -16036.031,E2 -16036.031} C_VEL
LIN {X 0,Y 305.026,Z 660.92,A -85,B 0,C 180,E1 -16039.716,E2 -16039.716} C_VEL
LIN {X 0,Y 306.08,Z 664.116,A -85,B 0,C 180,E1 -16039.979,E2 -16039.979} C_VEL
LIN {X 0,Y 310.052,Z 675.68,A -85,B 0,C 180,E1 -16041.073,E2 -16041.073} C_VEL
LIN {X 0,Y 313.006,Z 687.18,A -85,B 0,C 180,E1 -16042.266,E2 -16042.266} C_VEL
LIN {X 0,Y 314.605,Z 696.837,A -85,B 0,C 180,E1 -16043.361,E2 -16043.361} C_VEL
LIN {X 0,Y 314.611,Z 701.176,A -85,B 0,C 180,E1 -16043.851,E2 -16043.851} C_VEL
LIN {X 0,Y 313.067,Z 711.45,A -85,B 0,C 180,E1 -16045.052,E2 -16045.052} C_VEL
LIN {X 0,Y 311.38,Z 721.774,A -85,B 0,C 180,E1 -16046.561,E2 -16046.561} C_VEL
LIN {X 0,Y 309.771,Z 730.374,A -85,B 0,C 180,E1 -16048.107,E2 -16048.107} C_VEL
LIN {X 0,Y 308.063,Z 739.402,A -85,B 0,C 180,E1 -16050.126,E2 -16050.126} C_VEL
LIN {X 0,Y 306.595,Z 747.116,A -85,B 0,C 180,E1 -16052.318,E2 -16052.318} C_VEL
LIN {X 0,Y 305.402,Z 753.259,A -85,B 0,C 180,E1 -16054.579,E2 -16054.579} C_VEL
LIN {X 0,Y 304.564,Z 757.938,A -85,B 0,C 180,E1 -16056.868,E2 -16056.868} C_VEL
LIN {X 0,Y 304.143,Z 760.519,A -85,B 0,C 180,E1 -16058.602,E2 -16058.602} C_VEL
LIN {X 0,Y 303.738,Z 762.437,A -85,B 0,C 180,E1 -16060.382,E2 -16060.382} C_VEL
LIN {X 0,Y 303.537,Z 763.643,A -85,B 0,C 180,E1 -16062.19,E2 -16062.19} C_VEL
LIN {X 0,Y 303.397,Z 764.079,A -85,B 0,C 180,E1 -16064.102,E2 -16064.102} C_VEL
LIN {X 0,Y 303.369,Z 763.702,A -85,B 0,C 180,E1 -16065.973,E2 -16065.973} C_VEL
LIN {X 0,Y 303.511,Z 762.565,A -85,B 0,C 180,E1 -16067.815,E2 -16067.815} C_VEL
LIN {X 0,Y 303.729,Z 760.479,A -85,B 0,C 180,E1 -16069.782,E2 -16069.782} C_VEL
LIN {X 0,Y 304.087,Z 757.348,A -85,B 0,C 180,E1 -16071.795,E2 -16071.795} C_VEL
LIN {X 0,Y 304.59,Z 752.994,A -85,B 0,C 180,E1 -16073.86,E2 -16073.86} C_VEL
LIN {X 0,Y 305.259,Z 747.192,A -85,B 0,C 180,E1 -16075.979,E2 -16075.979} C_VEL
LIN {X 0,Y 306.335,Z 739.608,A -85,B 0,C 180,E1 -16078.151,E2 -16078.151} C_VEL
LIN {X 0,Y 307.537,Z 731.093,A -85,B 0,C 180,E1 -16080.072,E2 -16080.072} C_VEL
LIN {X 0,Y 308.737,Z 722.29,A -85,B 0,C 180,E1 -16081.687,E2 -16081.687} C_VEL
LIN {X 0,Y 310.077,Z 711.987,A -85,B 0,C 180,E1 -16083.226,E2 -16083.226} C_VEL
LIN {X 0,Y 311.432,Z 700.256,A -85,B 0,C 180,E1 -16084.61,E2 -16084.61} C_VEL
LIN {X 0,Y 311.745,Z 694.696,A -85,B 0,C 180,E1 -16085.172,E2 -16085.172} C_VEL
LIN {X 0,Y 309.849,Z 683.155,A -85,B 0,C 180,E1 -16086.294,E2 -16086.294} C_VEL
LIN {X 0,Y 307.161,Z 670.55,A -85,B 0,C 180,E1 -16087.288,E2 -16087.288} C_VEL
LIN {X 0,Y 304.386,Z 659.392,A -85,B 0,C 180,E1 -16088.009,E2 -16088.009} C_VEL
LIN {X 0,Y 304.653,Z 656.024,A -85,B 0,C 180,E1 -16091.157,E2 -16091.157} C_VEL
LIN {X 0,Y 305.057,Z 651.642,A -85,B 0,C 180,E1 -16095.378,E2 -16095.378} C_VEL
LIN {X 0,Y 305.398,Z 647.596,A -85,B 0,C 180,E1 -16099.391,E2 -16099.391} C_VEL
LIN {X 0,Y 305.577,Z 646.423,A -85,B 0,C 180,E1 -16100.735,E2 -16100.735} C_VEL
LIN {X 0,Y 305.835,Z 646.388,A -85,B 0,C 180,E1 -16103.402,E2 -16103.402} C_VEL
LIN {X 0,Y 305.889,Z 646.38,A -85,B 0,C 180,E1 -16107.366,E2 -16107.366} C_VEL
LIN {X 0,Y 306.059,Z 646.358,A -85,B 0,C 180,E1 -16109.999,E2 -16109.999} C_VEL
LIN {X 0,Y 305.889,Z 646.381,A -85,B 0,C 180,E1 -16112.633,E2 -16112.633} C_VEL
LIN {X 0,Y 305.775,Z 646.397,A -85,B 0,C 180,E1 -16116.598,E2 -16116.598} C_VEL
LIN {X 0,Y 305.489,Z 646.431,A -85,B 0,C 180,E1 -16119.267,E2 -16119.267} C_VEL
LIN {X 0,Y 304.967,Z 646.582,A -85,B 0,C 180,E1 -16122.307,E2 -16122.307} C_VEL
LIN {X 0,Y 304.561,Z 651.532,A -85,B 0,C 180,E1 -16126.075,E2 -16126.075} C_VEL
LIN {X 0,Y 304.391,Z 655.2,A -85,B 0,C 180,E1 -16128.858,E2 -16128.858} C_VEL
LIN {X 0,Y 304.25,Z 658.174,A -85,B 0,C 180,E1 -16131.112,E2 -16131.112} C_VEL
LIN {X 0,Y 307.689,Z 672.455,A -85,B 0,C 180,E1 -16132.022,E2 -16132.022} C_VEL
LIN {X 0,Y 310.024,Z 684.157,A -85,B 0,C 180,E1 -16132.961,E2 -16132.961} C_VEL
LIN {X 0,Y 311.712,Z 694.197,A -85,B 0,C 180,E1 -16133.943,E2 -16133.943} C_VEL
LIN {X 0,Y 311.048,Z 702.764,A -85,B 0,C 180,E1 -16134.82,E2 -16134.82} C_VEL
LIN {X 0,Y 309.816,Z 712.943,A -85,B 0,C 180,E1 -16136.072,E2 -16136.072} C_VEL
LIN {X 0,Y 308.402,Z 723.977,A -85,B 0,C 180,E1 -16137.777,E2 -16137.777} C_VEL
LIN {X 0,Y 307.068,Z 733.311,A -85,B 0,C 180,E1 -16139.573,E2 -16139.573} C_VEL
LIN {X 0,Y 306.023,Z 740.92,A -85,B 0,C 180,E1 -16141.397,E2 -16141.397} C_VEL
LIN {X 0,Y 305.072,Z 748.164,A -85,B 0,C 180,E1 -16143.565,E2 -16143.565} C_VEL
LIN {X 0,Y 304.506,Z 752.62,A -85,B 0,C 180,E1 -16145.239,E2 -16145.239} C_VEL
LIN {X 0,Y 303.938,Z 757.409,A -85,B 0,C 180,E1 -16147.537,E2 -16147.537} C_VEL
LIN {X 0,Y 303.733,Z 759.214,A -85,B 0,C 180,E1 -16148.663,E2 -16148.663} C_VEL
LIN {X 0,Y 303.435,Z 761.404,A -85,B 0,C 180,E1 -16150.429,E2 -16150.429} C_VEL
LIN {X 0,Y 303.343,Z 762.847,A -85,B 0,C 180,E1 -16152.212,E2 -16152.212} C_VEL
LIN {X 0,Y 303.304,Z 763.59,A -85,B 0,C 180,E1 -16154.084,E2 -16154.084} C_VEL
LIN {X 0,Y 303.4,Z 763.537,A -85,B 0,C 180,E1 -16155.979,E2 -16155.979} C_VEL
LIN {X 0,Y 303.572,Z 762.691,A -85,B 0,C 180,E1 -16157.826,E2 -16157.826} C_VEL
LIN {X 0,Y 304.057,Z 759.925,A -85,B 0,C 180,E1 -16160.587,E2 -16160.587} C_VEL
LIN {X 0,Y 304.583,Z 757.023,A -85,B 0,C 180,E1 -16162.448,E2 -16162.448} C_VEL
LIN {X 0,Y 305.562,Z 751.791,A -85,B 0,C 180,E1 -16164.9,E2 -16164.9} C_VEL
LIN {X 0,Y 306.814,Z 744.89,A -85,B 0,C 180,E1 -16167.275,E2 -16167.275} C_VEL
LIN {X 0,Y 308.137,Z 738.061,A -85,B 0,C 180,E1 -16169.125,E2 -16169.125} C_VEL
LIN {X 0,Y 309.771,Z 729.539,A -85,B 0,C 180,E1 -16170.991,E2 -16170.991} C_VEL
LIN {X 0,Y 311.405,Z 720.254,A -85,B 0,C 180,E1 -16172.623,E2 -16172.623} C_VEL
LIN {X 0,Y 313.192,Z 709.129,A -85,B 0,C 180,E1 -16174.197,E2 -16174.197} C_VEL
LIN {X 0,Y 313.54,Z 706.761,A -85,B 0,C 180,E1 -16174.48,E2 -16174.48} C_VEL
LIN {X 0,Y 313.595,Z 703.553,A -85,B 0,C 180,E1 -16174.889,E2 -16174.889} C_VEL
LIN {X 0,Y 312.512,Z 698.918,A -85,B 0,C 180,E1 -16175.54,E2 -16175.54} C_VEL
LIN {X 0,Y 310.58,Z 694.546,A -85,B 0,C 180,E1 -16176.202,E2 -16176.202} C_VEL
LIN {X 0,Y 306.22,Z 685.488,A -85,B 0,C 180,E1 -16177.489,E2 -16177.489} C_VEL
LIN {X 0,Y 305.218,Z 682.135,A -85,B 0,C 180,E1 -16177.872,E2 -16177.872} C_VEL
LIN {X 0,Y 301.466,Z 669.29,A -85,B 0,C 180,E1 -16179.175,E2 -16179.175} C_VEL
LIN {X 0,Y 298.013,Z 659.953,A -85,B 0,C 180,E1 -16180.035,E2 -16180.035} C_VEL
LIN {X 0,Y 297.902,Z 659.278,A -85,B 0,C 180,E1 -16180.133,E2 -16180.133} C_VEL
LIN {X 0,Y 298.18,Z 654.942,A -85,B 0,C 180,E1 -16183.57,E2 -16183.57} C_VEL
LIN {X 0,Y 298.52,Z 651.412,A -85,B 0,C 180,E1 -16186.383,E2 -16186.383} C_VEL
LIN {X 0,Y 298.518,Z 647.578,A -85,B 0,C 180,E1 -16189.487,E2 -16189.487} C_VEL
LIN {X 0,Y 298.504,Z 647.303,A -85,B 0,C 180,E1 -16189.829,E2 -16189.829} C_VEL
LIN {X 0,Y 298.778,Z 647.272,A -85,B 0,C 180,E1 -16193.246,E2 -16193.246} C_VEL
LIN {X 0,Y 298.922,Z 647.251,A -85,B 0,C 180,E1 -16198.653,E2 -16198.653} C_VEL
LIN {X 0,Y 298.922,Z 647.252,A -85,B 0,C 180,E1 -16201.347,E2 -16201.347} C_VEL
LIN {X 0,Y 298.794,Z 647.268,A -85,B 0,C 180,E1 -16206.754,E2 -16206.754} C_VEL
LIN {X 0,Y 298.677,Z 647.28,A -85,B 0,C 180,E1 -16209.481,E2 -16209.481} C_VEL
LIN {X 0,Y 298.549,Z 647.297,A -85,B 0,C 180,E1 -16213.616,E2 -16213.616} C_VEL
LIN {X 0,Y 298.545,Z 647.296,A -85,B 0,C 180,E1 -16216.409,E2 -16216.409} C_VEL
LIN {X 0,Y 298.508,Z 647.302,A -85,B 0,C 180,E1 -16219.655,E2 -16219.655} C_VEL
LIN {X 0,Y 298.454,Z 647.307,A -85,B 0,C 180,E1 -16223.598,E2 -16223.598} C_VEL
LIN {X 0,Y 298.486,Z 647.303,A -85,B 0,C 180,E1 -16226.575,E2 -16226.575} C_VEL
LIN {X 0,Y 298.418,Z 647.314,A -85,B 0,C 180,E1 -16229.641,E2 -16229.641} C_VEL
LIN {X 0,Y 298.392,Z 647.316,A -85,B 0,C 180,E1 -16232.801,E2 -16232.801} C_VEL
LIN {X 0,Y 298.444,Z 647.311,A -85,B 0,C 180,E1 -16236.808,E2 -16236.808} C_VEL
LIN {X 0,Y 298.385,Z 647.319,A -85,B 0,C 180,E1 -16241.088,E2 -16241.088} C_VEL
LIN {X 0,Y 298.386,Z 647.319,A -85,B 0,C 180,E1 -16245.042,E2 -16245.042} C_VEL
LIN {X 0,Y 298.558,Z 648.037,A -85,B 0,C 180,E1 -16245.886,E2 -16245.886} C_VEL
LIN {X 0,Y 299.366,Z 652.697,A -85,B 0,C 180,E1 -16249.79,E2 -16249.79} C_VEL
LIN {X 0,Y 299.841,Z 656.033,A -85,B 0,C 180,E1 -16252.454,E2 -16252.454} C_VEL
LIN {X 0,Y 299.838,Z 659.541,A -85,B 0,C 180,E1 -16255.123,E2 -16255.123} C_VEL
LIN {X 0,Y 299.11,Z 664.733,A -85,B 0,C 180,E1 -16258.875,E2 -16258.875} C_VEL
LIN {X 0,Y 298.424,Z 670.093,A -85,B 0,C 180,E1 -16262.663,E2 -16262.663} C_VEL
LIN {X 0,Y 298.134,Z 672.332,A -85,B 0,C 180,E1 -16264.214,E2 -16264.214} C_VEL
LIN {X 0,Y 298.962,Z 675.678,A -85,B 0,C 180,E1 -16264.451,E2 -16264.451} C_VEL
LIN {X 0,Y 302.457,Z 688.539,A -85,B 0,C 180,E1 -16265.523,E2 -16265.523} C_VEL
LIN {X 0,Y 304.747,Z 701.196,A -85,B 0,C 180,E1 -16266.711,E2 -16266.711} C_VEL
LIN {X 0,Y 305.671,Z 712.125,A -85,B 0,C 180,E1 -16267.867,E2 -16267.867} C_VEL
LIN {X 0,Y 305.972,Z 721.117,A -85,B 0,C 180,E1 -16268.968,E2 -16268.968} C_VEL
LIN {X 0,Y 304.25,Z 732.237,A -85,B 0,C 180,E1 -16270.432,E2 -16270.432} C_VEL
LIN {X 0,Y 302.522,Z 742.169,A -85,B 0,C 180,E1 -16272.073,E2 -16272.073} C_VEL
LIN {X 0,Y 300.977,Z 750.33,A -85,B 0,C 180,E1 -16273.728,E2 -16273.728} C_VEL
LIN {X 0,Y 299.554,Z 758.358,A -85,B 0,C 180,E1 -16275.739,E2 -16275.739} C_VEL
LIN {X 0,Y 298.275,Z 764.841,A -85,B 0,C 180,E1 -16277.758,E2 -16277.758} C_VEL
LIN {X 0,Y 297.477,Z 769.993,A -85,B 0,C 180,E1 -16279.795,E2 -16279.795} C_VEL
LIN {X 0,Y 296.94,Z 774.001,A -85,B 0,C 180,E1 -16281.837,E2 -16281.837} C_VEL
LIN {X 0,Y 296.6,Z 777.733,A -85,B 0,C 180,E1 -16284.562,E2 -16284.562} C_VEL
LIN {X 0,Y 296.535,Z 780.434,A -85,B 0,C 180,E1 -16287.284,E2 -16287.284} C_VEL
LIN {X 0,Y 296.494,Z 781.297,A -85,B 0,C 180,E1 -16288.642,E2 -16288.642} C_VEL
LIN {X 0,Y 296.521,Z 781.717,A -85,B 0,C 180,E1 -16290.001,E2 -16290.001} C_VEL
LIN {X 0,Y 296.492,Z 781.728,A -85,B 0,C 180,E1 -16291.359,E2 -16291.359} C_VEL
LIN {X 0,Y 296.533,Z 781.349,A -85,B 0,C 180,E1 -16292.717,E2 -16292.717} C_VEL
LIN {X 0,Y 296.54,Z 780.577,A -85,B 0,C 180,E1 -16294.078,E2 -16294.078} C_VEL
LIN {X 0,Y 296.593,Z 779.187,A -85,B 0,C 180,E1 -16295.602,E2 -16295.602} C_VEL
LIN {X 0,Y 296.972,Z 775.689,A -85,B 0,C 180,E1 -16298.164,E2 -16298.164} C_VEL
LIN {X 0,Y 297.505,Z 771.743,A -85,B 0,C 180,E1 -16300.206,E2 -16300.206} C_VEL
LIN {X 0,Y 298.347,Z 766.68,A -85,B 0,C 180,E1 -16302.241,E2 -16302.241} C_VEL
LIN {X 0,Y 299.65,Z 760.374,A -85,B 0,C 180,E1 -16304.257,E2 -16304.257} C_VEL
LIN {X 0,Y 301.171,Z 752.537,A -85,B 0,C 180,E1 -16306.262,E2 -16306.262} C_VEL
LIN {X 0,Y 302.878,Z 742.837,A -85,B 0,C 180,E1 -16308.256,E2 -16308.256} C_VEL
LIN {X 0,Y 304.75,Z 732.87,A -85,B 0,C 180,E1 -16309.887,E2 -16309.887} C_VEL
LIN {X 0,Y 306.591,Z 721.721,A -85,B 0,C 180,E1 -16311.341,E2 -16311.341} C_VEL
LIN {X 0,Y 306.245,Z 711.492,A -85,B 0,C 180,E1 -16312.577,E2 -16312.577} C_VEL
LIN {X 0,Y 304.808,Z 699.537,A -85,B 0,C 180,E1 -16313.864,E2 -16313.864} C_VEL
LIN {X 0,Y 302.298,Z 687.644,A -85,B 0,C 180,E1 -16315.006,E2 -16315.006} C_VEL
LIN {X 0,Y 298.482,Z 674.778,A -85,B 0,C 180,E1 -16316.108,E2 -16316.108} C_VEL
LIN {X 0,Y 298.444,Z 674.283,A -85,B 0,C 180,E1 -16316.165,E2 -16316.165} C_VEL
LIN {X 0,Y 299.089,Z 669.653,A -85,B 0,C 180,E1 -16319.608,E2 -16319.608} C_VEL
LIN {X 0,Y 299.69,Z 665.738,A -85,B 0,C 180,E1 -16322.641,E2 -16322.641} C_VEL
LIN {X 0,Y 300.209,Z 661.856,A -85,B 0,C 180,E1 -16325.822,E2 -16325.822} C_VEL
LIN {X 0,Y 300.265,Z 659.966,A -85,B 0,C 180,E1 -16327.486,E2 -16327.486} C_VEL
LIN {X 0,Y 299.917,Z 656.275,A -85,B 0,C 180,E1 -16331.006,E2 -16331.006} C_VEL
LIN {X 0,Y 299.346,Z 652.779,A -85,B 0,C 180,E1 -16334.776,E2 -16334.776} C_VEL
LIN {X 0,Y 299.034,Z 650.88,A -85,B 0,C 180,E1 -16337.034,E2 -16337.034} C_VEL
LIN {X 0,Y 298.512,Z 647.977,A -85,B 0,C 180,E1 -16340.981,E2 -16340.981} C_VEL
LIN {X 0,Y 298.41,Z 647.318,A -85,B 0,C 180,E1 -16342.241,E2 -16342.241} C_VEL
LIN {X 0,Y 298.41,Z 647.314,A -85,B 0,C 180,E1 -16345.581,E2 -16345.581} C_VEL
LIN {X 0,Y 298.394,Z 647.318,A -85,B 0,C 180,E1 -16348.791,E2 -16348.791} C_VEL
LIN {X 0,Y 298.459,Z 647.306,A -85,B 0,C 180,E1 -16351.904,E2 -16351.904} C_VEL
LIN {X 0,Y 298.485,Z 647.307,A -85,B 0,C 180,E1 -16354.924,E2 -16354.924} C_VEL
LIN {X 0,Y 298.452,Z 647.31,A -85,B 0,C 180,E1 -16359.315,E2 -16359.315} C_VEL
LIN {X 0,Y 298.54,Z 647.299,A -85,B 0,C 180,E1 -16362.179,E2 -16362.179} C_VEL
LIN {X 0,Y 298.595,Z 647.292,A -85,B 0,C 180,E1 -16364.995,E2 -16364.995} C_VEL
LIN {X 0,Y 298.596,Z 647.293,A -85,B 0,C 180,E1 -16369.147,E2 -16369.147} C_VEL
LIN {X 0,Y 298.76,Z 647.269,A -85,B 0,C 180,E1 -16371.886,E2 -16371.886} C_VEL
LIN {X 0,Y 298.662,Z 647.282,A -85,B 0,C 180,E1 -16374.599,E2 -16374.599} C_VEL
LIN {X 0,Y 298.926,Z 647.25,A -85,B 0,C 180,E1 -16378.653,E2 -16378.653} C_VEL
LIN {X 0,Y 299.012,Z 647.241,A -85,B 0,C 180,E1 -16380,E2 -16380} C_VEL
LIN {X 0,Y 299.052,Z 648.48,A -85,B 0,C 180,E1 -16382.694,E2 -16382.694} C_VEL
LIN {X 0,Y 299.252,Z 651.215,A -85,B 0,C 180,E1 -16386.838,E2 -16386.838} C_VEL
LIN {X 0,Y 299.229,Z 653.136,A -85,B 0,C 180,E1 -16389.463,E2 -16389.463} C_VEL
LIN {X 0,Y 298.674,Z 656.514,A -85,B 0,C 180,E1 -16393.61,E2 -16393.61} C_VEL
LIN {X 0,Y 298.146,Z 660.195,A -85,B 0,C 180,E1 -16397.845,E2 -16397.845} C_VEL
LIN {X 0,Y 298.092,Z 661.255,A -85,B 0,C 180,E1 -16398.916,E2 -16398.916} C_VEL
LIN {X 0,Y 300.278,Z 667.391,A -85,B 0,C 180,E1 -16399.483,E2 -16399.483} C_VEL
LIN {X 0,Y 303.901,Z 678.105,A -85,B 0,C 180,E1 -16400.578,E2 -16400.578} C_VEL
LIN {X 0,Y 306.474,Z 688.297,A -85,B 0,C 180,E1 -16401.702,E2 -16401.702} C_VEL
LIN {X 0,Y 308,Z 697.677,A -85,B 0,C 180,E1 -16402.825,E2 -16402.825} C_VEL
LIN {X 0,Y 308.258,Z 701.072,A -85,B 0,C 180,E1 -16403.248,E2 -16403.248} C_VEL
LIN {X 0,Y 306.552,Z 712.03,A -85,B 0,C 180,E1 -16404.553,E2 -16404.553} C_VEL
LIN {X 0,Y 304.685,Z 722.678,A -85,B 0,C 180,E1 -16406.158,E2 -16406.158} C_VEL
LIN {X 0,Y 302.812,Z 732.214,A -85,B 0,C 180,E1 -16407.954,E2 -16407.954} C_VEL
LIN {X 0,Y 301.267,Z 739.918,A -85,B 0,C 180,E1 -16409.752,E2 -16409.752} C_VEL
LIN {X 0,Y 299.688,Z 747.587,A -85,B 0,C 180,E1 -16412.007,E2 -16412.007} C_VEL
LIN {X 0,Y 298.404,Z 753.893,A -85,B 0,C 180,E1 -16414.42,E2 -16414.42} C_VEL
LIN {X 0,Y 297.558,Z 758.149,A -85,B 0,C 180,E1 -16416.578,E2 -16416.578} C_VEL
LIN {X 0,Y 297.033,Z 761.134,A -85,B 0,C 180,E1 -16418.666,E2 -16418.666} C_VEL
LIN {X 0,Y 296.608,Z 763.064,A -85,B 0,C 180,E1 -16420.691,E2 -16420.691} C_VEL
LIN {X 0,Y 296.338,Z 764.246,A -85,B 0,C 180,E1 -16423.454,E2 -16423.454} C_VEL
LIN {X 0,Y 296.259,Z 764.12,A -85,B 0,C 180,E1 -16425.372,E2 -16425.372} C_VEL
LIN {X 0,Y 296.369,Z 763.152,A -85,B 0,C 180,E1 -16427.318,E2 -16427.318} C_VEL
LIN {X 0,Y 296.571,Z 761.278,A -85,B 0,C 180,E1 -16429.317,E2 -16429.317} C_VEL
LIN {X 0,Y 296.941,Z 758.417,A -85,B 0,C 180,E1 -16431.357,E2 -16431.357} C_VEL
LIN {X 0,Y 297.468,Z 753.644,A -85,B 0,C 180,E1 -16433.796,E2 -16433.796} C_VEL
LIN {X 0,Y 298.193,Z 747.752,A -85,B 0,C 180,E1 -16436.03,E2 -16436.03} C_VEL
LIN {X 0,Y 299.172,Z 740.903,A -85,B 0,C 180,E1 -16438.076,E2 -16438.076} C_VEL
LIN {X 0,Y 300.317,Z 732.986,A -85,B 0,C 180,E1 -16439.983,E2 -16439.983} C_VEL
LIN {X 0,Y 301.738,Z 723.237,A -85,B 0,C 180,E1 -16441.858,E2 -16441.858} C_VEL
LIN {X 0,Y 303.176,Z 712.613,A -85,B 0,C 180,E1 -16443.497,E2 -16443.497} C_VEL
LIN {X 0,Y 304.37,Z 702.724,A -85,B 0,C 180,E1 -16444.728,E2 -16444.728} C_VEL
LIN {X 0,Y 304.988,Z 697.158,A -85,B 0,C 180,E1 -16445.316,E2 -16445.316} C_VEL
LIN {X 0,Y 303.448,Z 686.615,A -85,B 0,C 180,E1 -16446.407,E2 -16446.407} C_VEL
LIN {X 0,Y 300.716,Z 673.215,A -85,B 0,C 180,E1 -16447.546,E2 -16447.546} C_VEL
LIN {X 0,Y 297.329,Z 659.591,A -85,B 0,C 180,E1 -16448.462,E2 -16448.462} C_VEL
LIN {X 0,Y 297.638,Z 655.789,A -85,B 0,C 180,E1 -16452.123,E2 -16452.123} C_VEL
LIN {X 0,Y 298.084,Z 651.492,A -85,B 0,C 180,E1 -16456.362,E2 -16456.362} C_VEL
LIN {X 0,Y 298.504,Z 647.304,A -85,B 0,C 180,E1 -16460.66,E2 -16460.66} C_VEL
LIN {X 0,Y 298.777,Z 647.268,A -85,B 0,C 180,E1 -16463.245,E2 -16463.245} C_VEL
LIN {X 0,Y 298.927,Z 647.249,A -85,B 0,C 180,E1 -16468.652,E2 -16468.652} C_VEL
LIN {X 0,Y 298.927,Z 647.247,A -85,B 0,C 180,E1 -16471.347,E2 -16471.347} C_VEL
LIN {X 0,Y 298.643,Z 647.284,A -85,B 0,C 180,E1 -16475.401,E2 -16475.401} C_VEL
LIN {X 0,Y 298.606,Z 647.285,A -85,B 0,C 180,E1 -16478.118,E2 -16478.118} C_VEL
LIN {X 0,Y 297.936,Z 647.422,A -85,B 0,C 180,E1 -16482.257,E2 -16482.257} C_VEL
LIN {X 0,Y 297.479,Z 652.904,A -85,B 0,C 180,E1 -16486.469,E2 -16486.469} C_VEL
LIN {X 0,Y 297.208,Z 658.321,A -85,B 0,C 180,E1 -16490.639,E2 -16490.639} C_VEL
LIN {X 0,Y 300.725,Z 672.778,A -85,B 0,C 180,E1 -16491.597,E2 -16491.597} C_VEL
LIN {X 0,Y 303.225,Z 685.506,A -85,B 0,C 180,E1 -16492.663,E2 -16492.663} C_VEL
LIN {X 0,Y 304.904,Z 696.503,A -85,B 0,C 180,E1 -16493.788,E2 -16493.788} C_VEL
LIN {X 0,Y 303.724,Z 707.214,A -85,B 0,C 180,E1 -16494.971,E2 -16494.971} C_VEL
LIN {X 0,Y 302.359,Z 717.564,A -85,B 0,C 180,E1 -16496.393,E2 -16496.393} C_VEL
LIN {X 0,Y 300.891,Z 728.175,A -85,B 0,C 180,E1 -16498.227,E2 -16498.227} C_VEL
LIN {X 0,Y 299.631,Z 736.835,A -85,B 0,C 180,E1 -16500.088,E2 -16500.088} C_VEL
LIN {X 0,Y 298.601,Z 744.234,A -85,B 0,C 180,E1 -16502.079,E2 -16502.079} C_VEL
LIN {X 0,Y 297.731,Z 750.771,A -85,B 0,C 180,E1 -16504.291,E2 -16504.291} C_VEL
LIN {X 0,Y 297.076,Z 755.723,A -85,B 0,C 180,E1 -16506.453,E2 -16506.453} C_VEL
LIN {X 0,Y 296.646,Z 759.339,A -85,B 0,C 180,E1 -16508.572,E2 -16508.572} C_VEL
LIN {X 0,Y 296.314,Z 761.802,A -85,B 0,C 180,E1 -16510.625,E2 -16510.625} C_VEL
LIN {X 0,Y 296.218,Z 763.285,A -85,B 0,C 180,E1 -16512.65,E2 -16512.65} C_VEL
LIN {X 0,Y 296.255,Z 763.845,A -85,B 0,C 180,E1 -16515.371,E2 -16515.371} C_VEL
LIN {X 0,Y 296.412,Z 763.285,A -85,B 0,C 180,E1 -16517.307,E2 -16517.307} C_VEL
LIN {X 0,Y 296.684,Z 761.867,A -85,B 0,C 180,E1 -16519.29,E2 -16519.29} C_VEL
LIN {X 0,Y 297.159,Z 759.515,A -85,B 0,C 180,E1 -16521.302,E2 -16521.302} C_VEL
LIN {X 0,Y 298.003,Z 755.058,A -85,B 0,C 180,E1 -16523.872,E2 -16523.872} C_VEL
LIN {X 0,Y 299.044,Z 749.862,A -85,B 0,C 180,E1 -16526.071,E2 -16526.071} C_VEL
LIN {X 0,Y 300.411,Z 742.981,A -85,B 0,C 180,E1 -16528.311,E2 -16528.311} C_VEL
LIN {X 0,Y 302.198,Z 734.353,A -85,B 0,C 180,E1 -16530.5,E2 -16530.5} C_VEL
LIN {X 0,Y 303.875,Z 725.55,A -85,B 0,C 180,E1 -16532.276,E2 -16532.276} C_VEL
LIN {X 0,Y 305.689,Z 715.485,A -85,B 0,C 180,E1 -16533.904,E2 -16533.904} C_VEL
LIN {X 0,Y 307.464,Z 704.37,A -85,B 0,C 180,E1 -16535.345,E2 -16535.345} C_VEL
LIN {X 0,Y 308.09,Z 699.801,A -85,B 0,C 180,E1 -16535.845,E2 -16535.845} C_VEL
LIN {X 0,Y 306.716,Z 689.484,A -85,B 0,C 180,E1 -16537.074,E2 -16537.074} C_VEL
LIN {X 0,Y 305.218,Z 682.135,A -85,B 0,C 180,E1 -16537.872,E2 -16537.872} C_VEL
LIN {X 0,Y 303.846,Z 679.075,A -85,B 0,C 180,E1 -16538.266,E2 -16538.266} C_VEL
LIN {X 0,Y 299.996,Z 675.119,A -85,B 0,C 180,E1 -16538.992,E2 -16538.992} C_VEL
LIN {X 0,Y 295.887,Z 671.21,A -85,B 0,C 180,E1 -16539.717,E2 -16539.717} C_VEL
LIN {X 0,Y 294.109,Z 668.192,A -85,B 0,C 180,E1 -16540.102,E2 -16540.102} C_VEL
LIN {X 0,Y 291.078,Z 660.102,A -85,B 0,C 180,E1 -16540.889,E2 -16540.889} C_VEL
LIN {X 0,Y 290.996,Z 659.516,A -85,B 0,C 180,E1 -16540.952,E2 -16540.952} C_VEL
LIN {X 0,Y 291.374,Z 654.835,A -85,B 0,C 180,E1 -16544.751,E2 -16544.751} C_VEL
LIN {X 0,Y 291.598,Z 651.476,A -85,B 0,C 180,E1 -16547.472,E2 -16547.472} C_VEL
LIN {X 0,Y 291.52,Z 648.173,A -85,B 0,C 180,E1 -16550.284,E2 -16550.284} C_VEL
LIN {X 0,Y 291.723,Z 648.151,A -85,B 0,C 180,E1 -16553.081,E2 -16553.081} C_VEL
LIN {X 0,Y 291.888,Z 648.127,A -85,B 0,C 180,E1 -16558.62,E2 -16558.62} C_VEL
LIN {X 0,Y 291.888,Z 648.128,A -85,B 0,C 180,E1 -16561.38,E2 -16561.38} C_VEL
LIN {X 0,Y 291.743,Z 648.146,A -85,B 0,C 180,E1 -16566.918,E2 -16566.918} C_VEL
LIN {X 0,Y 291.626,Z 648.158,A -85,B 0,C 180,E1 -16569.712,E2 -16569.712} C_VEL
LIN {X 0,Y 291.518,Z 648.171,A -85,B 0,C 180,E1 -16573.95,E2 -16573.95} C_VEL
LIN {X 0,Y 291.483,Z 648.175,A -85,B 0,C 180,E1 -16576.818,E2 -16576.818} C_VEL
LIN {X 0,Y 291.447,Z 648.182,A -85,B 0,C 180,E1 -16579.875,E2 -16579.875} C_VEL
LIN {X 0,Y 291.397,Z 648.186,A -85,B 0,C 180,E1 -16584.206,E2 -16584.206} C_VEL
LIN {X 0,Y 291.42,Z 648.187,A -85,B 0,C 180,E1 -16587.272,E2 -16587.272} C_VEL
LIN {X 0,Y 291.334,Z 648.195,A -85,B 0,C 180,E1 -16590.437,E2 -16590.437} C_VEL
LIN {X 0,Y 291.342,Z 648.194,A -85,B 0,C 180,E1 -16593.699,E2 -16593.699} C_VEL
LIN {X 0,Y 291.373,Z 648.19,A -85,B 0,C 180,E1 -16597.255,E2 -16597.255} C_VEL
LIN {X 0,Y 291.33,Z 648.197,A -85,B 0,C 180,E1 -16600.643,E2 -16600.643} C_VEL
LIN {X 0,Y 291.364,Z 648.206,A -85,B 0,C 180,E1 -16605.02,E2 -16605.02} C_VEL
LIN {X 0,Y 292.021,Z 651.913,A -85,B 0,C 180,E1 -16608.251,E2 -16608.251} C_VEL
LIN {X 0,Y 292.694,Z 655.65,A -85,B 0,C 180,E1 -16611.37,E2 -16611.37} C_VEL
LIN {X 0,Y 292.861,Z 658.943,A -85,B 0,C 180,E1 -16613.982,E2 -16613.982} C_VEL
LIN {X 0,Y 292.313,Z 663.356,A -85,B 0,C 180,E1 -16617.298,E2 -16617.298} C_VEL
LIN {X 0,Y 291.597,Z 668.676,A -85,B 0,C 180,E1 -16621.182,E2 -16621.182} C_VEL
LIN {X 0,Y 291.198,Z 671.707,A -85,B 0,C 180,E1 -16623.351,E2 -16623.351} C_VEL
LIN {X 0,Y 292.055,Z 675.117,A -85,B 0,C 180,E1 -16623.613,E2 -16623.613} C_VEL
LIN {X 0,Y 295.476,Z 687.254,A -85,B 0,C 180,E1 -16624.668,E2 -16624.668} C_VEL
LIN {X 0,Y 297.767,Z 698.931,A -85,B 0,C 180,E1 -16625.802,E2 -16625.802} C_VEL
LIN {X 0,Y 298.965,Z 709.739,A -85,B 0,C 180,E1 -16626.974,E2 -16626.974} C_VEL
LIN {X 0,Y 299.353,Z 721.836,A -85,B 0,C 180,E1 -16628.48,E2 -16628.48} C_VEL
LIN {X 0,Y 297.596,Z 732.742,A -85,B 0,C 180,E1 -16629.976,E2 -16629.976} C_VEL
LIN {X 0,Y 295.77,Z 742.502,A -85,B 0,C 180,E1 -16631.649,E2 -16631.649} C_VEL
LIN {X 0,Y 294.141,Z 750.554,A -85,B 0,C 180,E1 -16633.339,E2 -16633.339} C_VEL
LIN {X 0,Y 292.669,Z 758.505,A -85,B 0,C 180,E1 -16635.396,E2 -16635.396} C_VEL
LIN {X 0,Y 291.316,Z 764.906,A -85,B 0,C 180,E1 -16637.46,E2 -16637.46} C_VEL
LIN {X 0,Y 290.469,Z 769.995,A -85,B 0,C 180,E1 -16639.546,E2 -16639.546} C_VEL
LIN {X 0,Y 289.889,Z 773.947,A -85,B 0,C 180,E1 -16641.637,E2 -16641.637} C_VEL
LIN {X 0,Y 289.639,Z 775.988,A -85,B 0,C 180,E1 -16643.032,E2 -16643.032} C_VEL
LIN {X 0,Y 289.447,Z 778.867,A -85,B 0,C 180,E1 -16645.823,E2 -16645.823} C_VEL
LIN {X 0,Y 289.462,Z 780.143,A -85,B 0,C 180,E1 -16647.217,E2 -16647.217} C_VEL
LIN {X 0,Y 289.416,Z 781.03,A -85,B 0,C 180,E1 -16648.609,E2 -16648.609} C_VEL
LIN {X 0,Y 289.438,Z 781.492,A -85,B 0,C 180,E1 -16650.001,E2 -16650.001} C_VEL
LIN {X 0,Y 289.414,Z 781.525,A -85,B 0,C 180,E1 -16651.392,E2 -16651.392} C_VEL
LIN {X 0,Y 289.439,Z 781.166,A -85,B 0,C 180,E1 -16652.784,E2 -16652.784} C_VEL
LIN {X 0,Y 289.444,Z 780.416,A -85,B 0,C 180,E1 -16654.178,E2 -16654.178} C_VEL
LIN {X 0,Y 289.517,Z 779.247,A -85,B 0,C 180,E1 -16655.573,E2 -16655.573} C_VEL
LIN {X 0,Y 289.781,Z 776.705,A -85,B 0,C 180,E1 -16657.666,E2 -16657.666} C_VEL
LIN {X 0,Y 290.279,Z 773.168,A -85,B 0,C 180,E1 -16659.758,E2 -16659.758} C_VEL
LIN {X 0,Y 291.098,Z 768.558,A -85,B 0,C 180,E1 -16661.843,E2 -16661.843} C_VEL
LIN {X 0,Y 292.513,Z 761.62,A -85,B 0,C 180,E1 -16664.257,E2 -16664.257} C_VEL
LIN {X 0,Y 294.103,Z 754.15,A -85,B 0,C 180,E1 -16666.307,E2 -16666.307} C_VEL
LIN {X 0,Y 295.501,Z 746.591,A -85,B 0,C 180,E1 -16668.011,E2 -16668.011} C_VEL
LIN {X 0,Y 297.294,Z 737.502,A -85,B 0,C 180,E1 -16669.687,E2 -16669.687} C_VEL
LIN {X 0,Y 299.189,Z 727.548,A -85,B 0,C 180,E1 -16671.172,E2 -16671.172} C_VEL
LIN {X 0,Y 299.994,Z 722.415,A -85,B 0,C 180,E1 -16671.834,E2 -16671.834} C_VEL
LIN {X 0,Y 299.73,Z 712.677,A -85,B 0,C 180,E1 -16673.076,E2 -16673.076} C_VEL
LIN {X 0,Y 298.371,Z 700.862,A -85,B 0,C 180,E1 -16674.412,E2 -16674.412} C_VEL
LIN {X 0,Y 296.043,Z 689.626,A -85,B 0,C 180,E1 -16675.563,E2 -16675.563} C_VEL
LIN {X 0,Y 292.4,Z 677.218,A -85,B 0,C 180,E1 -16676.741,E2 -16676.741} C_VEL
LIN {X 0,Y 291.545,Z 674.079,A -85,B 0,C 180,E1 -16676.992,E2 -16676.992} C_VEL
LIN {X 0,Y 292.154,Z 669.733,A -85,B 0,C 180,E1 -16680.343,E2 -16680.343} C_VEL
LIN {X 0,Y 292.808,Z 665.801,A -85,B 0,C 180,E1 -16683.508,E2 -16683.508} C_VEL
LIN {X 0,Y 293.158,Z 663.549,A -85,B 0,C 180,E1 -16685.403,E2 -16685.403} C_VEL
LIN {X 0,Y 293.193,Z 660.1,A -85,B 0,C 180,E1 -16688.553,E2 -16688.553} C_VEL
LIN {X 0,Y 292.786,Z 656.49,A -85,B 0,C 180,E1 -16692.231,E2 -16692.231} C_VEL
LIN {X 0,Y 292.186,Z 653.057,A -85,B 0,C 180,E1 -16696.187,E2 -16696.187} C_VEL
LIN {X 0,Y 291.634,Z 649.912,A -85,B 0,C 180,E1 -16700.458,E2 -16700.458} C_VEL
LIN {X 0,Y 291.406,Z 648.336,A -85,B 0,C 180,E1 -16702.919,E2 -16702.919} C_VEL
LIN {X 0,Y 291.346,Z 648.193,A -85,B 0,C 180,E1 -16706.302,E2 -16706.302} C_VEL
LIN {X 0,Y 291.385,Z 648.189,A -85,B 0,C 180,E1 -16710.261,E2 -16710.261} C_VEL
LIN {X 0,Y 291.414,Z 648.184,A -85,B 0,C 180,E1 -16714.272,E2 -16714.272} C_VEL
LIN {X 0,Y 291.383,Z 648.191,A -85,B 0,C 180,E1 -16717.3,E2 -16717.3} C_VEL
LIN {X 0,Y 291.46,Z 648.18,A -85,B 0,C 180,E1 -16720.27,E2 -16720.27} C_VEL
LIN {X 0,Y 291.557,Z 648.169,A -85,B 0,C 180,E1 -16724.624,E2 -16724.624} C_VEL
LIN {X 0,Y 291.539,Z 648.172,A -85,B 0,C 180,E1 -16728.881,E2 -16728.881} C_VEL
LIN {X 0,Y 291.711,Z 648.147,A -85,B 0,C 180,E1 -16731.689,E2 -16731.689} C_VEL
LIN {X 0,Y 291.633,Z 648.157,A -85,B 0,C 180,E1 -16734.468,E2 -16734.468} C_VEL
LIN {X 0,Y 291.892,Z 648.127,A -85,B 0,C 180,E1 -16738.62,E2 -16738.62} C_VEL
LIN {X 0,Y 292,Z 648.32,A -85,B 0,C 180,E1 -16740,E2 -16740} C_VEL
LIN {X 0,Y 292.083,Z 649.903,A -85,B 0,C 180,E1 -16742.758,E2 -16742.758} C_VEL
LIN {X 0,Y 292.269,Z 652.553,A -85,B 0,C 180,E1 -16746.906,E2 -16746.906} C_VEL
LIN {X 0,Y 292.202,Z 654.556,A -85,B 0,C 180,E1 -16749.693,E2 -16749.693} C_VEL
LIN {X 0,Y 291.601,Z 657.942,A -85,B 0,C 180,E1 -16753.947,E2 -16753.947} C_VEL
LIN {X 0,Y 291.108,Z 661.399,A -85,B 0,C 180,E1 -16758.019,E2 -16758.019} C_VEL
LIN {X 0,Y 292.229,Z 664.684,A -85,B 0,C 180,E1 -16758.349,E2 -16758.349} C_VEL
LIN {X 0,Y 296.276,Z 675.675,A -85,B 0,C 180,E1 -16759.531,E2 -16759.531} C_VEL
LIN {X 0,Y 299.552,Z 687.543,A -85,B 0,C 180,E1 -16760.89,E2 -16760.89} C_VEL
LIN {X 0,Y 301.502,Z 698.556,A -85,B 0,C 180,E1 -16762.259,E2 -16762.259} C_VEL
LIN {X 0,Y 301.731,Z 702.614,A -85,B 0,C 180,E1 -16762.783,E2 -16762.783} C_VEL
LIN {X 0,Y 299.936,Z 713.406,A -85,B 0,C 180,E1 -16764.134,E2 -16764.134} C_VEL
LIN {X 0,Y 298.171,Z 722.939,A -85,B 0,C 180,E1 -16765.624,E2 -16765.624} C_VEL
LIN {X 0,Y 296.094,Z 732.772,A -85,B 0,C 180,E1 -16767.52,E2 -16767.52} C_VEL
LIN {X 0,Y 294.531,Z 740.146,A -85,B 0,C 180,E1 -16769.286,E2 -16769.286} C_VEL
LIN {X 0,Y 292.932,Z 747.577,A -85,B 0,C 180,E1 -16771.509,E2 -16771.509} C_VEL
LIN {X 0,Y 291.661,Z 753.21,A -85,B 0,C 180,E1 -16773.657,E2 -16773.657} C_VEL
LIN {X 0,Y 290.59,Z 758.289,A -85,B 0,C 180,E1 -16776.221,E2 -16776.221} C_VEL
LIN {X 0,Y 290.056,Z 761.042,A -85,B 0,C 180,E1 -16778.16,E2 -16778.16} C_VEL
LIN {X 0,Y 289.481,Z 763.593,A -85,B 0,C 180,E1 -16780.958,E2 -16780.958} C_VEL
LIN {X 0,Y 289.263,Z 764.453,A -85,B 0,C 180,E1 -16783.206,E2 -16783.206} C_VEL
LIN {X 0,Y 289.174,Z 764.366,A -85,B 0,C 180,E1 -16785.185,E2 -16785.185} C_VEL
LIN {X 0,Y 289.271,Z 763.453,A -85,B 0,C 180,E1 -16787.134,E2 -16787.134} C_VEL
LIN {X 0,Y 289.447,Z 761.801,A -85,B 0,C 180,E1 -16789.036,E2 -16789.036} C_VEL
LIN {X 0,Y 289.921,Z 757.967,A -85,B 0,C 180,E1 -16791.825,E2 -16791.825} C_VEL
LIN {X 0,Y 290.362,Z 754.121,A -85,B 0,C 180,E1 -16793.794,E2 -16793.794} C_VEL
LIN {X 0,Y 291.21,Z 747.709,A -85,B 0,C 180,E1 -16796.284,E2 -16796.284} C_VEL
LIN {X 0,Y 292.273,Z 740.485,A -85,B 0,C 180,E1 -16798.466,E2 -16798.466} C_VEL
LIN {X 0,Y 293.629,Z 731.451,A -85,B 0,C 180,E1 -16800.615,E2 -16800.615} C_VEL
LIN {X 0,Y 295.107,Z 721.375,A -85,B 0,C 180,E1 -16802.523,E2 -16802.523} C_VEL
LIN {X 0,Y 296.655,Z 710.212,A -85,B 0,C 180,E1 -16804.192,E2 -16804.192} C_VEL
LIN {X 0,Y 298.114,Z 697.975,A -85,B 0,C 180,E1 -16805.634,E2 -16805.634} C_VEL
LIN {X 0,Y 296.518,Z 687.204,A -85,B 0,C 180,E1 -16806.793,E2 -16806.793} C_VEL
LIN {X 0,Y 293.836,Z 673.959,A -85,B 0,C 180,E1 -16807.962,E2 -16807.962} C_VEL
LIN {X 0,Y 290.546,Z 661.19,A -85,B 0,C 180,E1 -16808.865,E2 -16808.865} C_VEL
LIN {X 0,Y 290.297,Z 659.806,A -85,B 0,C 180,E1 -16808.938,E2 -16808.938} C_VEL
LIN {X 0,Y 290.528,Z 657.021,A -85,B 0,C 180,E1 -16811.67,E2 -16811.67} C_VEL
LIN {X 0,Y 291.003,Z 652.681,A -85,B 0,C 180,E1 -16816.024,E2 -16816.024} C_VEL
LIN {X 0,Y 291.477,Z 648.18,A -85,B 0,C 180,E1 -16820.703,E2 -16820.703} C_VEL
LIN {X 0,Y 291.722,Z 648.148,A -85,B 0,C 180,E1 -16823.081,E2 -16823.081} C_VEL
LIN {X 0,Y 291.893,Z 648.125,A -85,B 0,C 180,E1 -16828.62,E2 -16828.62} C_VEL
LIN {X 0,Y 291.893,Z 648.122,A -85,B 0,C 180,E1 -16831.379,E2 -16831.379} C_VEL
LIN {X 0,Y 291.609,Z 648.159,A -85,B 0,C 180,E1 -16835.531,E2 -16835.531} C_VEL
LIN {X 0,Y 291.537,Z 648.166,A -85,B 0,C 180,E1 -16838.316,E2 -16838.316} C_VEL
LIN {X 0,Y 290.889,Z 648.266,A -85,B 0,C 180,E1 -16842.204,E2 -16842.204} C_VEL
LIN {X 0,Y 290.508,Z 652.401,A -85,B 0,C 180,E1 -16845.432,E2 -16845.432} C_VEL
LIN {X 0,Y 290.195,Z 658.279,A -85,B 0,C 180,E1 -16850.003,E2 -16850.003} C_VEL
LIN {X 0,Y 290.197,Z 658.636,A -85,B 0,C 180,E1 -16850.188,E2 -16850.188} C_VEL
LIN {X 0,Y 293.422,Z 671.873,A -85,B 0,C 180,E1 -16851.055,E2 -16851.055} C_VEL
LIN {X 0,Y 296.071,Z 684.634,A -85,B 0,C 180,E1 -16852.137,E2 -16852.137} C_VEL
LIN {X 0,Y 297.869,Z 695.604,A -85,B 0,C 180,E1 -16853.278,E2 -16853.278} C_VEL
LIN {X 0,Y 297.903,Z 699.004,A -85,B 0,C 180,E1 -16853.643,E2 -16853.643} C_VEL
LIN {X 0,Y 296.432,Z 710.884,A -85,B 0,C 180,E1 -16855.073,E2 -16855.073} C_VEL
LIN {X 0,Y 295.055,Z 720.766,A -85,B 0,C 180,E1 -16856.559,E2 -16856.559} C_VEL
LIN {X 0,Y 293.646,Z 730.557,A -85,B 0,C 180,E1 -16858.391,E2 -16858.391} C_VEL
LIN {X 0,Y 292.364,Z 738.859,A -85,B 0,C 180,E1 -16860.318,E2 -16860.318} C_VEL
LIN {X 0,Y 291.356,Z 746.1,A -85,B 0,C 180,E1 -16862.407,E2 -16862.407} C_VEL
LIN {X 0,Y 290.499,Z 752.22,A -85,B 0,C 180,E1 -16864.658,E2 -16864.658} C_VEL
LIN {X 0,Y 289.87,Z 756.826,A -85,B 0,C 180,E1 -16866.86,E2 -16866.86} C_VEL
LIN {X 0,Y 289.444,Z 760.334,A -85,B 0,C 180,E1 -16869.146,E2 -16869.146} C_VEL
LIN {X 0,Y 289.177,Z 762.4,A -85,B 0,C 180,E1 -16871.113,E2 -16871.113} C_VEL
LIN {X 0,Y 289.121,Z 763.677,A -85,B 0,C 180,E1 -16873.177,E2 -16873.177} C_VEL
LIN {X 0,Y 289.154,Z 764.076,A -85,B 0,C 180,E1 -16875.182,E2 -16875.182} C_VEL
LIN {X 0,Y 289.312,Z 763.658,A -85,B 0,C 180,E1 -16877.142,E2 -16877.142} C_VEL
LIN {X 0,Y 289.546,Z 762.457,A -85,B 0,C 180,E1 -16879.053,E2 -16879.053} C_VEL
LIN {X 0,Y 290.257,Z 759.285,A -85,B 0,C 180,E1 -16881.871,E2 -16881.871} C_VEL
LIN {X 0,Y 291.243,Z 754.474,A -85,B 0,C 180,E1 -16884.609,E2 -16884.609} C_VEL
LIN {X 0,Y 292.408,Z 748.989,A -85,B 0,C 180,E1 -16886.863,E2 -16886.863} C_VEL
LIN {X 0,Y 293.687,Z 742.944,A -85,B 0,C 180,E1 -16888.823,E2 -16888.823} C_VEL
LIN {X 0,Y 295.332,Z 735.491,A -85,B 0,C 180,E1 -16890.766,E2 -16890.766} C_VEL
LIN {X 0,Y 297.209,Z 726.138,A -85,B 0,C 180,E1 -16892.732,E2 -16892.732} C_VEL
LIN {X 0,Y 299.152,Z 715.955,A -85,B 0,C 180,E1 -16894.425,E2 -16894.425} C_VEL
LIN {X 0,Y 301.014,Z 705.022,A -85,B 0,C 180,E1 -16895.883,E2 -16895.883} C_VEL
LIN {X 0,Y 301.545,Z 701.028,A -85,B 0,C 180,E1 -16896.34,E2 -16896.34} C_VEL
LIN {X 0,Y 300.192,Z 690.674,A -85,B 0,C 180,E1 -16897.639,E2 -16897.639} C_VEL
LIN {X 0,Y 297.962,Z 680.434,A -85,B 0,C 180,E1 -16898.804,E2 -16898.804} C_VEL
LIN {X 0,Y 294.278,Z 668.611,A -85,B 0,C 180,E1 -16900.058,E2 -16900.058} C_VEL
LIN {X 0,Y 294.109,Z 668.192,A -85,B 0,C 180,E1 -16900.102,E2 -16900.102} C_VEL
LIN {X 0,Y 292.295,Z 665.128,A -85,B 0,C 180,E1 -16900.504,E2 -16900.504} C_VEL
LIN {X 0,Y 289.903,Z 662.787,A -85,B 0,C 180,E1 -16900.992,E2 -16900.992} C_VEL
LIN {X 0,Y 286.713,Z 660.483,A -85,B 0,C 180,E1 -16901.768,E2 -16901.768} C_VEL
LIN {X 0,Y 284.678,Z 658.961,A -85,B 0,C 180,E1 -16902.581,E2 -16902.581} C_VEL
LIN {X 0,Y 284.171,Z 658.068,A -85,B 0,C 180,E1 -16903.229,E2 -16903.229} C_VEL
LIN {X 0,Y 284.608,Z 653.336,A -85,B 0,C 180,E1 -16907.159,E2 -16907.159} C_VEL
LIN {X 0,Y 284.571,Z 649.409,A -85,B 0,C 180,E1 -16910.543,E2 -16910.543} C_VEL
LIN {X 0,Y 284.587,Z 649.039,A -85,B 0,C 180,E1 -16911.042,E2 -16911.042} C_VEL
LIN {X 0,Y 284.594,Z 649.039,A -85,B 0,C 180,E1 -16914.331,E2 -16914.331} C_VEL
LIN {X 0,Y 284.854,Z 649.003,A -85,B 0,C 180,E1 -16918.586,E2 -16918.586} C_VEL
LIN {X 0,Y 284.854,Z 649.004,A -85,B 0,C 180,E1 -16921.414,E2 -16921.414} C_VEL
LIN {X 0,Y 284.695,Z 649.023,A -85,B 0,C 180,E1 -16927.09,E2 -16927.09} C_VEL
LIN {X 0,Y 284.563,Z 649.038,A -85,B 0,C 180,E1 -16929.955,E2 -16929.955} C_VEL
LIN {X 0,Y 284.478,Z 649.047,A -85,B 0,C 180,E1 -16934.303,E2 -16934.303} C_VEL
LIN {X 0,Y 284.422,Z 649.057,A -85,B 0,C 180,E1 -16937.249,E2 -16937.249} C_VEL
LIN {X 0,Y 284.375,Z 649.064,A -85,B 0,C 180,E1 -16940.242,E2 -16940.242} C_VEL
LIN {X 0,Y 284.366,Z 649.061,A -85,B 0,C 180,E1 -16943.876,E2 -16943.876} C_VEL
LIN {X 0,Y 284.394,Z 649.061,A -85,B 0,C 180,E1 -16947.174,E2 -16947.174} C_VEL
LIN {X 0,Y 284.293,Z 649.071,A -85,B 0,C 180,E1 -16951.275,E2 -16951.275} C_VEL
LIN {X 0,Y 284.338,Z 649.065,A -85,B 0,C 180,E1 -16955.349,E2 -16955.349} C_VEL
LIN {X 0,Y 284.309,Z 649.069,A -85,B 0,C 180,E1 -16958.17,E2 -16958.17} C_VEL
LIN {X 0,Y 284.266,Z 649.074,A -85,B 0,C 180,E1 -16962.125,E2 -16962.125} C_VEL
LIN {X 0,Y 284.347,Z 649.262,A -85,B 0,C 180,E1 -16964.92,E2 -16964.92} C_VEL
LIN {X 0,Y 285.017,Z 653.007,A -85,B 0,C 180,E1 -16968.26,E2 -16968.26} C_VEL
LIN {X 0,Y 285.611,Z 656.359,A -85,B 0,C 180,E1 -16971.13,E2 -16971.13} C_VEL
LIN {X 0,Y 285.81,Z 660.18,A -85,B 0,C 180,E1 -16974.239,E2 -16974.239} C_VEL
LIN {X 0,Y 285.284,Z 664.023,A -85,B 0,C 180,E1 -16977.183,E2 -16977.183} C_VEL
LIN {X 0,Y 284.531,Z 669.391,A -85,B 0,C 180,E1 -16981.207,E2 -16981.207} C_VEL
LIN {X 0,Y 284.328,Z 671.225,A -85,B 0,C 180,E1 -16982.447,E2 -16982.447} C_VEL
LIN {X 0,Y 285.309,Z 674.791,A -85,B 0,C 180,E1 -16982.732,E2 -16982.732} C_VEL
LIN {X 0,Y 288.666,Z 686.694,A -85,B 0,C 180,E1 -16983.829,E2 -16983.829} C_VEL
LIN {X 0,Y 291.209,Z 698.979,A -85,B 0,C 180,E1 -16985.088,E2 -16985.088} C_VEL
LIN {X 0,Y 292.376,Z 709.009,A -85,B 0,C 180,E1 -16986.217,E2 -16986.217} C_VEL
LIN {X 0,Y 292.742,Z 721.224,A -85,B 0,C 180,E1 -16987.784,E2 -16987.784} C_VEL
LIN {X 0,Y 292.261,Z 726.345,A -85,B 0,C 180,E1 -16988.488,E2 -16988.488} C_VEL
LIN {X 0,Y 290.349,Z 736.366,A -85,B 0,C 180,E1 -16990.008,E2 -16990.008} C_VEL
LIN {X 0,Y 288.425,Z 745.702,A -85,B 0,C 180,E1 -16991.778,E2 -16991.778} C_VEL
LIN {X 0,Y 286.833,Z 753.623,A -85,B 0,C 180,E1 -16993.635,E2 -16993.635} C_VEL
LIN {X 0,Y 285.309,Z 760.916,A -85,B 0,C 180,E1 -16995.74,E2 -16995.74} C_VEL
LIN {X 0,Y 284.056,Z 766.793,A -85,B 0,C 180,E1 -16997.861,E2 -16997.861} C_VEL
LIN {X 0,Y 283.223,Z 771.439,A -85,B 0,C 180,E1 -16999.998,E2 -16999.998} C_VEL
LIN {X 0,Y 282.689,Z 774.985,A -85,B 0,C 180,E1 -17002.142,E2 -17002.142} C_VEL
LIN {X 0,Y 282.407,Z 777.748,A -85,B 0,C 180,E1 -17004.529,E2 -17004.529} C_VEL
LIN {X 0,Y 282.368,Z 779.852,A -85,B 0,C 180,E1 -17007.147,E2 -17007.147} C_VEL
LIN {X 0,Y 282.34,Z 780.762,A -85,B 0,C 180,E1 -17008.574,E2 -17008.574} C_VEL
LIN {X 0,Y 282.358,Z 781.265,A -85,B 0,C 180,E1 -17010.001,E2 -17010.001} C_VEL
LIN {X 0,Y 282.337,Z 781.322,A -85,B 0,C 180,E1 -17011.427,E2 -17011.427} C_VEL
LIN {X 0,Y 282.347,Z 780.985,A -85,B 0,C 180,E1 -17012.854,E2 -17012.854} C_VEL
LIN {X 0,Y 282.41,Z 779.338,A -85,B 0,C 180,E1 -17015.476,E2 -17015.476} C_VEL
LIN {X 0,Y 282.603,Z 777.559,A -85,B 0,C 180,E1 -17017.143,E2 -17017.143} C_VEL
LIN {X 0,Y 283.061,Z 774.417,A -85,B 0,C 180,E1 -17019.288,E2 -17019.288} C_VEL
LIN {X 0,Y 283.81,Z 770.231,A -85,B 0,C 180,E1 -17021.427,E2 -17021.427} C_VEL
LIN {X 0,Y 285.093,Z 763.873,A -85,B 0,C 180,E1 -17023.908,E2 -17023.908} C_VEL
LIN {X 0,Y 286.727,Z 756.997,A -85,B 0,C 180,E1 -17026.007,E2 -17026.007} C_VEL
LIN {X 0,Y 288.087,Z 750.096,A -85,B 0,C 180,E1 -17027.747,E2 -17027.747} C_VEL
LIN {X 0,Y 289.805,Z 741.771,A -85,B 0,C 180,E1 -17029.479,E2 -17029.479} C_VEL
LIN {X 0,Y 291.928,Z 731.664,A -85,B 0,C 180,E1 -17031.169,E2 -17031.169} C_VEL
LIN {X 0,Y 293.416,Z 723.187,A -85,B 0,C 180,E1 -17032.349,E2 -17032.349} C_VEL
LIN {X 0,Y 293.205,Z 713.761,A -85,B 0,C 180,E1 -17033.608,E2 -17033.608} C_VEL
LIN {X 0,Y 291.894,Z 701.816,A -85,B 0,C 180,E1 -17035.034,E2 -17035.034} C_VEL
LIN {X 0,Y 289.783,Z 691.298,A -85,B 0,C 180,E1 -17036.188,E2 -17036.188} C_VEL
LIN {X 0,Y 286.306,Z 679.319,A -85,B 0,C 180,E1 -17037.407,E2 -17037.407} C_VEL
LIN {X 0,Y 284.689,Z 674.111,A -85,B 0,C 180,E1 -17037.888,E2 -17037.888} C_VEL
